LIN {X 0,Y 418.224,Z 205.699,A -85,B 0,C 180,E1 -10122.319,E2 -10122.319} C_VEL
LIN {X 0,Y 418.235,Z 205.697,A -85,B 0,C 180,E1 -10125.108,E2 -10125.108} C_VEL
LIN {X 0,Y 418.224,Z 205.697,A -85,B 0,C 180,E1 -10127.764,E2 -10127.764} C_VEL
LIN {X 0,Y 418.241,Z 205.702,A -85,B 0,C 180,E1 -10131.556,E2 -10131.556} C_VEL
LIN {X 0,Y 418.228,Z 205.712,A -85,B 0,C 180,E1 -10132.974,E2 -10132.974} C_VEL
LIN {X 0,Y 423.651,Z 221.501,A -85,B 0,C 180,E1 -10135.664,E2 -10135.664} C_VEL
LIN {X 0,Y 426.35,Z 230.16,A -85,B 0,C 180,E1 -10137.028,E2 -10137.028} C_VEL
LIN {X 0,Y 433.959,Z 245.967,A -85,B 0,C 180,E1 -10138.023,E2 -10138.023} C_VEL
LIN {X 0,Y 437.099,Z 265.296,A -85,B 0,C 180,E1 -10138.671,E2 -10138.671} C_VEL
LIN {X 0,Y 433.148,Z 437.708,A -85,B 0,C 180,E1 -10141.719,E2 -10141.719} C_VEL
LIN {X 0,Y 432.221,Z 453.77,A -85,B 0,C 180,E1 -10142.161,E2 -10142.161} C_VEL
LIN {X 0,Y 431.126,Z 469.58,A -85,B 0,C 180,E1 -10142.775,E2 -10142.775} C_VEL
LIN {X 0,Y 429.85,Z 484.792,A -85,B 0,C 180,E1 -10143.541,E2 -10143.541} C_VEL
LIN {X 0,Y 428.366,Z 499.512,A -85,B 0,C 180,E1 -10144.469,E2 -10144.469} C_VEL
LIN {X 0,Y 426.802,Z 513.668,A -85,B 0,C 180,E1 -10145.559,E2 -10145.559} C_VEL
LIN {X 0,Y 425.173,Z 527.972,A -85,B 0,C 180,E1 -10146.883,E2 -10146.883} C_VEL
LIN {X 0,Y 423.786,Z 539.159,A -85,B 0,C 180,E1 -10148.092,E2 -10148.092} C_VEL
LIN {X 0,Y 422.302,Z 550.643,A -85,B 0,C 180,E1 -10149.543,E2 -10149.543} C_VEL
LIN {X 0,Y 420.912,Z 562.204,A -85,B 0,C 180,E1 -10151.25,E2 -10151.25} C_VEL
LIN {X 0,Y 419.814,Z 572.306,A -85,B 0,C 180,E1 -10152.997,E2 -10152.997} C_VEL
LIN {X 0,Y 418.809,Z 581.69,A -85,B 0,C 180,E1 -10154.922,E2 -10154.922} C_VEL
LIN {X 0,Y 418.116,Z 589.681,A -85,B 0,C 180,E1 -10156.878,E2 -10156.878} C_VEL
LIN {X 0,Y 417.594,Z 596.384,A -85,B 0,C 180,E1 -10158.839,E2 -10158.839} C_VEL
LIN {X 0,Y 417.237,Z 601.811,A -85,B 0,C 180,E1 -10160.79,E2 -10160.79} C_VEL
LIN {X 0,Y 417.142,Z 605.169,A -85,B 0,C 180,E1 -10162.252,E2 -10162.252} C_VEL
LIN {X 0,Y 417.065,Z 608.619,A -85,B 0,C 180,E1 -10164.195,E2 -10164.195} C_VEL
LIN {X 0,Y 416.965,Z 611.127,A -85,B 0,C 180,E1 -10166.132,E2 -10166.132} C_VEL
LIN {X 0,Y 417.062,Z 612.548,A -85,B 0,C 180,E1 -10168.066,E2 -10168.066} C_VEL
LIN {X 0,Y 416.999,Z 613.082,A -85,B 0,C 180,E1 -10169.998,E2 -10169.998} C_VEL
LIN {X 0,Y 417.061,Z 612.552,A -85,B 0,C 180,E1 -10171.929,E2 -10171.929} C_VEL
LIN {X 0,Y 416.964,Z 611.13,A -85,B 0,C 180,E1 -10173.863,E2 -10173.863} C_VEL
LIN {X 0,Y 417.135,Z 607.929,A -85,B 0,C 180,E1 -10176.259,E2 -10176.259} C_VEL
LIN {X 0,Y 417.18,Z 604.08,A -85,B 0,C 180,E1 -10178.23,E2 -10178.23} C_VEL
LIN {X 0,Y 417.386,Z 599.247,A -85,B 0,C 180,E1 -10180.181,E2 -10180.181} C_VEL
LIN {X 0,Y 417.854,Z 593.155,A -85,B 0,C 180,E1 -10182.134,E2 -10182.134} C_VEL
LIN {X 0,Y 418.386,Z 585.778,A -85,B 0,C 180,E1 -10184.094,E2 -10184.094} C_VEL
LIN {X 0,Y 419.336,Z 576.968,A -85,B 0,C 180,E1 -10186.051,E2 -10186.051} C_VEL
LIN {X 0,Y 420.386,Z 566.446,A -85,B 0,C 180,E1 -10188.013,E2 -10188.013} C_VEL
LIN {X 0,Y 421.704,Z 555.505,A -85,B 0,C 180,E1 -10189.72,E2 -10189.72} C_VEL
LIN {X 0,Y 422.98,Z 544.609,A -85,B 0,C 180,E1 -10191.182,E2 -10191.182} C_VEL
LIN {X 0,Y 424.434,Z 531.99,A -85,B 0,C 180,E1 -10192.639,E2 -10192.639} C_VEL
LIN {X 0,Y 426.083,Z 518.332,A -85,B 0,C 180,E1 -10193.961,E2 -10193.961} C_VEL
LIN {X 0,Y 427.557,Z 505.031,A -85,B 0,C 180,E1 -10195.037,E2 -10195.037} C_VEL
LIN {X 0,Y 429.007,Z 490.343,A -85,B 0,C 180,E1 -10196.032,E2 -10196.032} C_VEL
LIN {X 0,Y 430.365,Z 474.899,A -85,B 0,C 180,E1 -10196.878,E2 -10196.878} C_VEL
LIN {X 0,Y 431.56,Z 458.018,A -85,B 0,C 180,E1 -10197.584,E2 -10197.584} C_VEL
LIN {X 0,Y 432.467,Z 442.335,A -85,B 0,C 180,E1 -10198.048,E2 -10198.048} C_VEL
LIN {X 0,Y 433.152,Z 419.903,A -85,B 0,C 180,E1 -10198.483,E2 -10198.483} C_VEL
LIN {X 0,Y 436.397,Z 265.424,A -85,B 0,C 180,E1 -10201.171,E2 -10201.171} C_VEL
LIN {X 0,Y 432.877,Z 244.923,A -85,B 0,C 180,E1 -10201.839,E2 -10201.839} C_VEL
LIN {X 0,Y 426.312,Z 230.881,A -85,B 0,C 180,E1 -10202.655,E2 -10202.655} C_VEL
LIN {X 0,Y 421.2,Z 214.684,A -85,B 0,C 180,E1 -10205.156,E2 -10205.156} C_VEL
LIN {X 0,Y 418.222,Z 205.707,A -85,B 0,C 180,E1 -10206.617,E2 -10206.617} C_VEL
LIN {X 0,Y 418.225,Z 205.697,A -85,B 0,C 180,E1 -10209.68,E2 -10209.68} C_VEL
LIN {X 0,Y 418.208,Z 205.699,A -85,B 0,C 180,E1 -10212.318,E2 -10212.318} C_VEL
LIN {X 0,Y 418.217,Z 205.698,A -85,B 0,C 180,E1 -10215.107,E2 -10215.107} C_VEL
LIN {X 0,Y 418.235,Z 205.7,A -85,B 0,C 180,E1 -10217.767,E2 -10217.767} C_VEL
LIN {X 0,Y 418.243,Z 205.697,A -85,B 0,C 180,E1 -10220.615,E2 -10220.615} C_VEL
LIN {X 0,Y 418.22,Z 205.694,A -85,B 0,C 180,E1 -10223.974,E2 -10223.974} C_VEL
LIN {X 0,Y 418.23,Z 205.691,A -85,B 0,C 180,E1 -10227.154,E2 -10227.154} C_VEL
LIN {X 0,Y 418.24,Z 205.704,A -85,B 0,C 180,E1 -10230.894,E2 -10230.894} C_VEL
LIN {X 0,Y 418.241,Z 205.683,A -85,B 0,C 180,E1 -10234.094,E2 -10234.094} C_VEL
LIN {X 0,Y 418.245,Z 205.697,A -85,B 0,C 180,E1 -10237.536,E2 -10237.536} C_VEL
LIN {X 0,Y 418.286,Z 205.673,A -85,B 0,C 180,E1 -10240.365,E2 -10240.365} C_VEL
LIN {X 0,Y 418.285,Z 205.693,A -85,B 0,C 180,E1 -10243.404,E2 -10243.404} C_VEL
LIN {X 0,Y 418.323,Z 205.665,A -85,B 0,C 180,E1 -10246.993,E2 -10246.993} C_VEL
LIN {X 0,Y 418.33,Z 205.681,A -85,B 0,C 180,E1 -10250.329,E2 -10250.329} C_VEL
LIN {X 0,Y 418.463,Z 205.666,A -85,B 0,C 180,E1 -10253.249,E2 -10253.249} C_VEL
LIN {X 0,Y 418.312,Z 205.667,A -85,B 0,C 180,E1 -10255.182,E2 -10255.182} C_VEL
LIN {X 0,Y 418.513,Z 205.648,A -85,B 0,C 180,E1 -10258.076,E2 -10258.076} C_VEL
LIN {X 0,Y 418.64,Z 205.645,A -85,B 0,C 180,E1 -10260,E2 -10260} C_VEL
LIN {X 0,Y 418.478,Z 205.661,A -85,B 0,C 180,E1 -10262.888,E2 -10262.888} C_VEL
LIN {X 0,Y 418.461,Z 205.67,A -85,B 0,C 180,E1 -10266.752,E2 -10266.752} C_VEL
LIN {X 0,Y 418.31,Z 205.684,A -85,B 0,C 180,E1 -10269.673,E2 -10269.673} C_VEL
LIN {X 0,Y 418.315,Z 205.682,A -85,B 0,C 180,E1 -10273.002,E2 -10273.002} C_VEL
LIN {X 0,Y 418.291,Z 205.687,A -85,B 0,C 180,E1 -10276.74,E2 -10276.74} C_VEL
LIN {X 0,Y 418.242,Z 205.684,A -85,B 0,C 180,E1 -10279.792,E2 -10279.792} C_VEL
LIN {X 0,Y 418.211,Z 205.702,A -85,B 0,C 180,E1 -10282.738,E2 -10282.738} C_VEL
LIN {X 0,Y 418.244,Z 205.683,A -85,B 0,C 180,E1 -10285.906,E2 -10285.906} C_VEL
LIN {X 0,Y 418.24,Z 205.697,A -85,B 0,C 180,E1 -10289.165,E2 -10289.165} C_VEL
LIN {X 0,Y 418.234,Z 205.686,A -85,B 0,C 180,E1 -10292.847,E2 -10292.847} C_VEL
LIN {X 0,Y 418.223,Z 205.705,A -85,B 0,C 180,E1 -10296.241,E2 -10296.241} C_VEL
LIN {X 0,Y 418.222,Z 205.686,A -85,B 0,C 180,E1 -10299.686,E2 -10299.686} C_VEL
LIN {X 0,Y 418.21,Z 205.706,A -85,B 0,C 180,E1 -10302.324,E2 -10302.324} C_VEL
LIN {X 0,Y 418.218,Z 205.687,A -85,B 0,C 180,E1 -10305.112,E2 -10305.112} C_VEL
LIN {X 0,Y 418.218,Z 205.702,A -85,B 0,C 180,E1 -10307.769,E2 -10307.769} C_VEL
LIN {X 0,Y 418.233,Z 205.693,A -85,B 0,C 180,E1 -10311.561,E2 -10311.561} C_VEL
LIN {X 0,Y 418.248,Z 205.688,A -85,B 0,C 180,E1 -10315.162,E2 -10315.162} C_VEL
LIN {X 0,Y 418.235,Z 205.698,A -85,B 0,C 180,E1 -10317.475,E2 -10317.475} C_VEL
LIN {X 0,Y 418.256,Z 205.694,A -85,B 0,C 180,E1 -10320.9,E2 -10320.9} C_VEL
LIN {X 0,Y 418.228,Z 205.696,A -85,B 0,C 180,E1 -10324.097,E2 -10324.097} C_VEL
LIN {X 0,Y 418.227,Z 205.697,A -85,B 0,C 180,E1 -10327.267,E2 -10327.267} C_VEL
LIN {X 0,Y 418.28,Z 205.691,A -85,B 0,C 180,E1 -10330.367,E2 -10330.367} C_VEL
LIN {X 0,Y 418.277,Z 205.693,A -85,B 0,C 180,E1 -10333.406,E2 -10333.406} C_VEL
LIN {X 0,Y 418.347,Z 205.686,A -85,B 0,C 180,E1 -10337.002,E2 -10337.002} C_VEL
LIN {X 0,Y 418.336,Z 205.686,A -85,B 0,C 180,E1 -10340.331,E2 -10340.331} C_VEL
LIN {X 0,Y 418.455,Z 205.75,A -85,B 0,C 180,E1 -10343.108,E2 -10343.108} C_VEL
LIN {X 0,Y 419.99,Z 210.519,A -85,B 0,C 180,E1 -10343.895,E2 -10343.895} C_VEL
LIN {X 0,Y 432.553,Z 235.499,A -85,B 0,C 180,E1 -10345.43,E2 -10345.43} C_VEL
LIN {X 0,Y 436.628,Z 244.415,A -85,B 0,C 180,E1 -10345.921,E2 -10345.921} C_VEL
LIN {X 0,Y 434.989,Z 317.307,A -85,B 0,C 180,E1 -10347.19,E2 -10347.19} C_VEL
LIN {X 0,Y 434.323,Z 323.153,A -85,B 0,C 180,E1 -10347.252,E2 -10347.252} C_VEL
LIN {X 0,Y 428.84,Z 342.222,A -85,B 0,C 180,E1 -10347.211,E2 -10347.211} C_VEL
LIN {X 0,Y 428.073,Z 348.075,A -85,B 0,C 180,E1 -10347.266,E2 -10347.266} C_VEL
LIN {X 0,Y 426.561,Z 416.445,A -85,B 0,C 180,E1 -10348.498,E2 -10348.498} C_VEL
LIN {X 0,Y 425.738,Z 433.559,A -85,B 0,C 180,E1 -10348.997,E2 -10348.997} C_VEL
LIN {X 0,Y 424.731,Z 449.304,A -85,B 0,C 180,E1 -10349.647,E2 -10349.647} C_VEL
LIN {X 0,Y 423.415,Z 464.949,A -85,B 0,C 180,E1 -10350.478,E2 -10350.478} C_VEL
LIN {X 0,Y 422.031,Z 479.6,A -85,B 0,C 180,E1 -10351.449,E2 -10351.449} C_VEL
LIN {X 0,Y 420.402,Z 494.314,A -85,B 0,C 180,E1 -10352.637,E2 -10352.637} C_VEL
LIN {X 0,Y 418.776,Z 507.961,A -85,B 0,C 180,E1 -10353.972,E2 -10353.972} C_VEL
LIN {X 0,Y 417.194,Z 520.585,A -85,B 0,C 180,E1 -10355.433,E2 -10355.433} C_VEL
LIN {X 0,Y 415.669,Z 532.421,A -85,B 0,C 180,E1 -10357.043,E2 -10357.043} C_VEL
LIN {X 0,Y 414.256,Z 543.314,A -85,B 0,C 180,E1 -10358.785,E2 -10358.785} C_VEL
LIN {X 0,Y 412.951,Z 553.803,A -85,B 0,C 180,E1 -10360.792,E2 -10360.792} C_VEL
LIN {X 0,Y 411.963,Z 562.602,A -85,B 0,C 180,E1 -10362.815,E2 -10362.815} C_VEL
LIN {X 0,Y 411.195,Z 569.983,A -85,B 0,C 180,E1 -10364.857,E2 -10364.857} C_VEL
LIN {X 0,Y 410.629,Z 576.107,A -85,B 0,C 180,E1 -10366.917,E2 -10366.917} C_VEL
LIN {X 0,Y 410.268,Z 580.967,A -85,B 0,C 180,E1 -10368.996,E2 -10368.996} C_VEL
LIN {X 0,Y 409.941,Z 584.701,A -85,B 0,C 180,E1 -10371.103,E2 -10371.103} C_VEL
LIN {X 0,Y 409.767,Z 587.357,A -85,B 0,C 180,E1 -10373.235,E2 -10373.235} C_VEL
LIN {X 0,Y 409.684,Z 588.815,A -85,B 0,C 180,E1 -10375.397,E2 -10375.397} C_VEL
LIN {X 0,Y 409.726,Z 589.143,A -85,B 0,C 180,E1 -10377.591,E2 -10377.591} C_VEL
LIN {X 0,Y 409.785,Z 588.303,A -85,B 0,C 180,E1 -10379.827,E2 -10379.827} C_VEL
LIN {X 0,Y 409.913,Z 586.13,A -85,B 0,C 180,E1 -10382.108,E2 -10382.108} C_VEL
LIN {X 0,Y 410.164,Z 582.538,A -85,B 0,C 180,E1 -10384.434,E2 -10384.434} C_VEL
LIN {X 0,Y 410.493,Z 578.367,A -85,B 0,C 180,E1 -10386.419,E2 -10386.419} C_VEL
LIN {X 0,Y 411.054,Z 572.44,A -85,B 0,C 180,E1 -10388.627,E2 -10388.627} C_VEL
LIN {X 0,Y 411.708,Z 566.367,A -85,B 0,C 180,E1 -10390.443,E2 -10390.443} C_VEL
LIN {X 0,Y 412.67,Z 557.711,A -85,B 0,C 180,E1 -10392.608,E2 -10392.608} C_VEL
LIN {X 0,Y 413.94,Z 547.818,A -85,B 0,C 180,E1 -10394.652,E2 -10394.652} C_VEL
LIN {X 0,Y 415.348,Z 537.429,A -85,B 0,C 180,E1 -10396.459,E2 -10396.459} C_VEL
LIN {X 0,Y 416.979,Z 525.311,A -85,B 0,C 180,E1 -10398.23,E2 -10398.23} C_VEL
LIN {X 0,Y 418.469,Z 513.861,A -85,B 0,C 180,E1 -10399.646,E2 -10399.646} C_VEL
LIN {X 0,Y 420.165,Z 500.476,A -85,B 0,C 180,E1 -10401.059,E2 -10401.059} C_VEL
LIN {X 0,Y 421.909,Z 485.847,A -85,B 0,C 180,E1 -10402.347,E2 -10402.347} C_VEL
LIN {X 0,Y 423.488,Z 471.058,A -85,B 0,C 180,E1 -10403.42,E2 -10403.42} C_VEL
LIN {X 0,Y 424.824,Z 456.217,A -85,B 0,C 180,E1 -10404.286,E2 -10404.286} C_VEL
LIN {X 0,Y 426.038,Z 439.8,A -85,B 0,C 180,E1 -10405.037,E2 -10405.037} C_VEL
LIN {X 0,Y 426.972,Z 423.004,A -85,B 0,C 180,E1 -10405.599,E2 -10405.599} C_VEL
LIN {X 0,Y 427.604,Z 405.792,A -85,B 0,C 180,E1 -10405.978,E2 -10405.978} C_VEL
LIN {X 0,Y 431.375,Z 247.088,A -85,B 0,C 180,E1 -10408.816,E2 -10408.816} C_VEL
LIN {X 0,Y 422.843,Z 229.659,A -85,B 0,C 180,E1 -10409.944,E2 -10409.944} C_VEL
LIN {X 0,Y 414.377,Z 214.394,A -85,B 0,C 180,E1 -10411.094,E2 -10411.094} C_VEL
LIN {X 0,Y 412.834,Z 211.442,A -85,B 0,C 180,E1 -10411.323,E2 -10411.323} C_VEL
LIN {X 0,Y 411.25,Z 206.571,A -85,B 0,C 180,E1 -10412.279,E2 -10412.279} C_VEL
LIN {X 0,Y 411.215,Z 206.574,A -85,B 0,C 180,E1 -10415.783,E2 -10415.783} C_VEL
LIN {X 0,Y 411.199,Z 206.57,A -85,B 0,C 180,E1 -10418.965,E2 -10418.965} C_VEL
LIN {X 0,Y 411.255,Z 206.562,A -85,B 0,C 180,E1 -10422.084,E2 -10422.084} C_VEL
LIN {X 0,Y 411.261,Z 206.567,A -85,B 0,C 180,E1 -10425.147,E2 -10425.147} C_VEL
LIN {X 0,Y 411.284,Z 206.569,A -85,B 0,C 180,E1 -10428.167,E2 -10428.167} C_VEL
LIN {X 0,Y 411.426,Z 206.55,A -85,B 0,C 180,E1 -10432.206,E2 -10432.206} C_VEL
LIN {X 0,Y 411.474,Z 206.541,A -85,B 0,C 180,E1 -10434.117,E2 -10434.117} C_VEL
LIN {X 0,Y 411.51,Z 206.538,A -85,B 0,C 180,E1 -10438.042,E2 -10438.042} C_VEL
LIN {X 0,Y 411.639,Z 206.524,A -85,B 0,C 180,E1 -10439.999,E2 -10439.999} C_VEL
LIN {X 0,Y 411.455,Z 206.543,A -85,B 0,C 180,E1 -10442.937,E2 -10442.937} C_VEL
LIN {X 0,Y 411.464,Z 206.545,A -85,B 0,C 180,E1 -10445.882,E2 -10445.882} C_VEL
LIN {X 0,Y 411.319,Z 206.561,A -85,B 0,C 180,E1 -10448.845,E2 -10448.845} C_VEL
LIN {X 0,Y 411.283,Z 206.567,A -85,B 0,C 180,E1 -10451.832,E2 -10451.832} C_VEL
LIN {X 0,Y 411.259,Z 206.569,A -85,B 0,C 180,E1 -10454.852,E2 -10454.852} C_VEL
LIN {X 0,Y 411.245,Z 206.569,A -85,B 0,C 180,E1 -10457.915,E2 -10457.915} C_VEL
LIN {X 0,Y 411.196,Z 206.578,A -85,B 0,C 180,E1 -10461.034,E2 -10461.034} C_VEL
LIN {X 0,Y 411.218,Z 206.569,A -85,B 0,C 180,E1 -10464.215,E2 -10464.215} C_VEL
LIN {X 0,Y 411.26,Z 206.568,A -85,B 0,C 180,E1 -10467.477,E2 -10467.477} C_VEL
LIN {X 0,Y 411.189,Z 206.579,A -85,B 0,C 180,E1 -10470.847,E2 -10470.847} C_VEL
LIN {X 0,Y 411.193,Z 206.574,A -85,B 0,C 180,E1 -10474.334,E2 -10474.334} C_VEL
LIN {X 0,Y 411.192,Z 206.576,A -85,B 0,C 180,E1 -10477.973,E2 -10477.973} C_VEL
LIN {X 0,Y 411.161,Z 206.573,A -85,B 0,C 180,E1 -10481.227,E2 -10481.227} C_VEL
LIN {X 0,Y 411.175,Z 206.574,A -85,B 0,C 180,E1 -10484.49,E2 -10484.49} C_VEL
LIN {X 0,Y 411.165,Z 206.578,A -85,B 0,C 180,E1 -10488.192,E2 -10488.192} C_VEL
LIN {X 0,Y 411.197,Z 206.577,A -85,B 0,C 180,E1 -10491.832,E2 -10491.832} C_VEL
LIN {X 0,Y 411.219,Z 206.749,A -85,B 0,C 180,E1 -10492.365,E2 -10492.365} C_VEL
LIN {X 0,Y 416.965,Z 223.279,A -85,B 0,C 180,E1 -10495.269,E2 -10495.269} C_VEL
LIN {X 0,Y 419.14,Z 230.129,A -85,B 0,C 180,E1 -10496.353,E2 -10496.353} C_VEL
LIN {X 0,Y 427.046,Z 246.152,A -85,B 0,C 180,E1 -10497.422,E2 -10497.422} C_VEL
LIN {X 0,Y 428.433,Z 249.802,A -85,B 0,C 180,E1 -10497.619,E2 -10497.619} C_VEL
LIN {X 0,Y 431.099,Z 267.046,A -85,B 0,C 180,E1 -10498.201,E2 -10498.201} C_VEL
LIN {X 0,Y 426.953,Z 437.436,A -85,B 0,C 180,E1 -10501.254,E2 -10501.254} C_VEL
LIN {X 0,Y 425.967,Z 453.95,A -85,B 0,C 180,E1 -10501.716,E2 -10501.716} C_VEL
LIN {X 0,Y 424.822,Z 469.64,A -85,B 0,C 180,E1 -10502.337,E2 -10502.337} C_VEL
LIN {X 0,Y 423.497,Z 484.763,A -85,B 0,C 180,E1 -10503.113,E2 -10503.113} C_VEL
LIN {X 0,Y 421.832,Z 500.369,A -85,B 0,C 180,E1 -10504.115,E2 -10504.115} C_VEL
LIN {X 0,Y 420.112,Z 514.978,A -85,B 0,C 180,E1 -10505.276,E2 -10505.276} C_VEL
LIN {X 0,Y 418.429,Z 529.014,A -85,B 0,C 180,E1 -10506.62,E2 -10506.62} C_VEL
LIN {X 0,Y 416.945,Z 540.466,A -85,B 0,C 180,E1 -10507.898,E2 -10507.898} C_VEL
LIN {X 0,Y 415.348,Z 552.287,A -85,B 0,C 180,E1 -10509.443,E2 -10509.443} C_VEL
LIN {X 0,Y 413.918,Z 563.541,A -85,B 0,C 180,E1 -10511.178,E2 -10511.178} C_VEL
LIN {X 0,Y 412.789,Z 573.36,A -85,B 0,C 180,E1 -10512.95,E2 -10512.95} C_VEL
LIN {X 0,Y 411.749,Z 582.616,A -85,B 0,C 180,E1 -10514.91,E2 -10514.91} C_VEL
LIN {X 0,Y 410.989,Z 591.343,A -85,B 0,C 180,E1 -10517.154,E2 -10517.154} C_VEL
LIN {X 0,Y 410.324,Z 599.079,A -85,B 0,C 180,E1 -10519.637,E2 -10519.637} C_VEL
LIN {X 0,Y 410.079,Z 604.974,A -85,B 0,C 180,E1 -10522.118,E2 -10522.118} C_VEL
LIN {X 0,Y 409.979,Z 608.421,A -85,B 0,C 180,E1 -10524.094,E2 -10524.094} C_VEL
LIN {X 0,Y 409.883,Z 610.927,A -85,B 0,C 180,E1 -10526.065,E2 -10526.065} C_VEL
LIN {X 0,Y 409.971,Z 612.346,A -85,B 0,C 180,E1 -10528.033,E2 -10528.033} C_VEL
LIN {X 0,Y 409.921,Z 612.876,A -85,B 0,C 180,E1 -10529.998,E2 -10529.998} C_VEL
LIN {X 0,Y 409.988,Z 612.343,A -85,B 0,C 180,E1 -10531.962,E2 -10531.962} C_VEL
LIN {X 0,Y 409.881,Z 610.915,A -85,B 0,C 180,E1 -10533.93,E2 -10533.93} C_VEL
LIN {X 0,Y 410.037,Z 607.925,A -85,B 0,C 180,E1 -10536.222,E2 -10536.222} C_VEL
LIN {X 0,Y 410.091,Z 603.851,A -85,B 0,C 180,E1 -10538.373,E2 -10538.373} C_VEL
LIN {X 0,Y 410.322,Z 599.008,A -85,B 0,C 180,E1 -10540.358,E2 -10540.358} C_VEL
LIN {X 0,Y 410.836,Z 592.91,A -85,B 0,C 180,E1 -10542.344,E2 -10542.344} C_VEL
LIN {X 0,Y 411.388,Z 585.521,A -85,B 0,C 180,E1 -10544.339,E2 -10544.339} C_VEL
LIN {X 0,Y 412.409,Z 576.698,A -85,B 0,C 180,E1 -10546.328,E2 -10546.328} C_VEL
LIN {X 0,Y 413.495,Z 566.161,A -85,B 0,C 180,E1 -10548.324,E2 -10548.324} C_VEL
LIN {X 0,Y 414.919,Z 555.209,A -85,B 0,C 180,E1 -10550.056,E2 -10550.056} C_VEL
LIN {X 0,Y 416.271,Z 544.283,A -85,B 0,C 180,E1 -10551.54,E2 -10551.54} C_VEL
LIN {X 0,Y 417.832,Z 531.625,A -85,B 0,C 180,E1 -10553.018,E2 -10553.018} C_VEL
LIN {X 0,Y 419.506,Z 517.933,A -85,B 0,C 180,E1 -10554.361,E2 -10554.361} C_VEL
LIN {X 0,Y 421.228,Z 502.917,A -85,B 0,C 180,E1 -10555.578,E2 -10555.578} C_VEL
LIN {X 0,Y 422.756,Z 487.631,A -85,B 0,C 180,E1 -10556.593,E2 -10556.593} C_VEL
LIN {X 0,Y 424.19,Z 471.683,A -85,B 0,C 180,E1 -10557.435,E2 -10557.435} C_VEL
LIN {X 0,Y 425.317,Z 455.528,A -85,B 0,C 180,E1 -10558.091,E2 -10558.091} C_VEL
LIN {X 0,Y 426.294,Z 439.16,A -85,B 0,C 180,E1 -10558.558,E2 -10558.558} C_VEL
LIN {X 0,Y 427.391,Z 389.53,A -85,B 0,C 180,E1 -10559.459,E2 -10559.459} C_VEL
LIN {X 0,Y 430.199,Z 265.695,A -85,B 0,C 180,E1 -10561.644,E2 -10561.644} C_VEL
LIN {X 0,Y 427.058,Z 247.804,A -85,B 0,C 180,E1 -10562.247,E2 -10562.247} C_VEL
LIN {X 0,Y 418.931,Z 230.448,A -85,B 0,C 180,E1 -10563.305,E2 -10563.305} C_VEL
LIN {X 0,Y 413.857,Z 214.643,A -85,B 0,C 180,E1 -10565.82,E2 -10565.82} C_VEL
LIN {X 0,Y 411.188,Z 206.576,A -85,B 0,C 180,E1 -10567.184,E2 -10567.184} C_VEL
LIN {X 0,Y 411.159,Z 206.578,A -85,B 0,C 180,E1 -10570.502,E2 -10570.502} C_VEL
LIN {X 0,Y 411.152,Z 206.578,A -85,B 0,C 180,E1 -10573.131,E2 -10573.131} C_VEL
LIN {X 0,Y 411.15,Z 206.576,A -85,B 0,C 180,E1 -10575.878,E2 -10575.878} C_VEL
LIN {X 0,Y 411.177,Z 206.574,A -85,B 0,C 180,E1 -10578.763,E2 -10578.763} C_VEL
LIN {X 0,Y 411.178,Z 206.577,A -85,B 0,C 180,E1 -10582.025,E2 -10582.025} C_VEL
LIN {X 0,Y 411.179,Z 206.578,A -85,B 0,C 180,E1 -10585.664,E2 -10585.664} C_VEL
LIN {X 0,Y 411.161,Z 206.574,A -85,B 0,C 180,E1 -10589.151,E2 -10589.151} C_VEL
LIN {X 0,Y 411.23,Z 206.567,A -85,B 0,C 180,E1 -10592.521,E2 -10592.521} C_VEL
LIN {X 0,Y 411.2,Z 206.574,A -85,B 0,C 180,E1 -10595.783,E2 -10595.783} C_VEL
LIN {X 0,Y 411.208,Z 206.562,A -85,B 0,C 180,E1 -10598.967,E2 -10598.967} C_VEL
LIN {X 0,Y 411.221,Z 206.565,A -85,B 0,C 180,E1 -10602.084,E2 -10602.084} C_VEL
LIN {X 0,Y 411.231,Z 206.567,A -85,B 0,C 180,E1 -10605.147,E2 -10605.147} C_VEL
LIN {X 0,Y 411.269,Z 206.538,A -85,B 0,C 180,E1 -10608.167,E2 -10608.167} C_VEL
LIN {X 0,Y 411.411,Z 206.549,A -85,B 0,C 180,E1 -10612.186,E2 -10612.186} C_VEL
LIN {X 0,Y 411.459,Z 206.537,A -85,B 0,C 180,E1 -10614.118,E2 -10614.118} C_VEL
LIN {X 0,Y 411.482,Z 206.523,A -85,B 0,C 180,E1 -10618.043,E2 -10618.043} C_VEL
LIN {X 0,Y 411.61,Z 206.521,A -85,B 0,C 180,E1 -10620.001,E2 -10620.001} C_VEL
LIN {X 0,Y 411.434,Z 206.538,A -85,B 0,C 180,E1 -10622.938,E2 -10622.938} C_VEL
LIN {X 0,Y 411.425,Z 206.548,A -85,B 0,C 180,E1 -10626.868,E2 -10626.868} C_VEL
LIN {X 0,Y 411.262,Z 206.562,A -85,B 0,C 180,E1 -10629.84,E2 -10629.84} C_VEL
LIN {X 0,Y 411.275,Z 206.56,A -85,B 0,C 180,E1 -10633.105,E2 -10633.105} C_VEL
LIN {X 0,Y 411.235,Z 206.564,A -85,B 0,C 180,E1 -10636.871,E2 -10636.871} C_VEL
LIN {X 0,Y 411.202,Z 206.561,A -85,B 0,C 180,E1 -10639.989,E2 -10639.989} C_VEL
LIN {X 0,Y 411.176,Z 206.575,A -85,B 0,C 180,E1 -10643.15,E2 -10643.15} C_VEL
LIN {X 0,Y 411.212,Z 206.56,A -85,B 0,C 180,E1 -10646.383,E2 -10646.383} C_VEL
LIN {X 0,Y 411.175,Z 206.578,A -85,B 0,C 180,E1 -10649.715,E2 -10649.715} C_VEL
LIN {X 0,Y 411.183,Z 206.564,A -85,B 0,C 180,E1 -10653.159,E2 -10653.159} C_VEL
LIN {X 0,Y 411.171,Z 206.58,A -85,B 0,C 180,E1 -10656.555,E2 -10656.555} C_VEL
LIN {X 0,Y 411.187,Z 206.562,A -85,B 0,C 180,E1 -10659.73,E2 -10659.73} C_VEL
LIN {X 0,Y 411.155,Z 206.579,A -85,B 0,C 180,E1 -10663.137,E2 -10663.137} C_VEL
LIN {X 0,Y 411.15,Z 206.57,A -85,B 0,C 180,E1 -10665.884,E2 -10665.884} C_VEL
LIN {X 0,Y 411.142,Z 206.58,A -85,B 0,C 180,E1 -10668.776,E2 -10668.776} C_VEL
LIN {X 0,Y 411.18,Z 206.576,A -85,B 0,C 180,E1 -10672.029,E2 -10672.029} C_VEL
LIN {X 0,Y 411.195,Z 206.567,A -85,B 0,C 180,E1 -10675.67,E2 -10675.67} C_VEL
LIN {X 0,Y 411.18,Z 206.575,A -85,B 0,C 180,E1 -10679.156,E2 -10679.156} C_VEL
LIN {X 0,Y 411.181,Z 206.578,A -85,B 0,C 180,E1 -10682.521,E2 -10682.521} C_VEL
LIN {X 0,Y 411.198,Z 206.578,A -85,B 0,C 180,E1 -10685.786,E2 -10685.786} C_VEL
LIN {X 0,Y 411.192,Z 206.577,A -85,B 0,C 180,E1 -10688.969,E2 -10688.969} C_VEL
LIN {X 0,Y 411.227,Z 206.578,A -85,B 0,C 180,E1 -10692.087,E2 -10692.087} C_VEL
LIN {X 0,Y 411.231,Z 206.574,A -85,B 0,C 180,E1 -10695.149,E2 -10695.149} C_VEL
LIN {X 0,Y 411.283,Z 206.564,A -85,B 0,C 180,E1 -10698.17,E2 -10698.17} C_VEL
LIN {X 0,Y 411.318,Z 206.564,A -85,B 0,C 180,E1 -10701.157,E2 -10701.157} C_VEL
LIN {X 0,Y 411.414,Z 206.705,A -85,B 0,C 180,E1 -10702.584,E2 -10702.584} C_VEL
LIN {X 0,Y 412.733,Z 210.707,A -85,B 0,C 180,E1 -10703.263,E2 -10703.263} C_VEL
LIN {X 0,Y 426.594,Z 237.914,A -85,B 0,C 180,E1 -10704.998,E2 -10704.998} C_VEL
LIN {X 0,Y 430.444,Z 246.548,A -85,B 0,C 180,E1 -10705.479,E2 -10705.479} C_VEL
LIN {X 0,Y 428.073,Z 348.075,A -85,B 0,C 180,E1 -10707.266,E2 -10707.266} C_VEL
LIN {X 0,Y 427.334,Z 353.923,A -85,B 0,C 180,E1 -10707.324,E2 -10707.324} C_VEL
LIN {X 0,Y 421.952,Z 373.01,A -85,B 0,C 180,E1 -10707.294,E2 -10707.294} C_VEL
LIN {X 0,Y 421.182,Z 378.86,A -85,B 0,C 180,E1 -10707.351,E2 -10707.351} C_VEL
LIN {X 0,Y 420.232,Z 417.941,A -85,B 0,C 180,E1 -10708.086,E2 -10708.086} C_VEL
LIN {X 0,Y 419.394,Z 434.723,A -85,B 0,C 180,E1 -10708.592,E2 -10708.592} C_VEL
LIN {X 0,Y 418.374,Z 449.581,A -85,B 0,C 180,E1 -10709.22,E2 -10709.22} C_VEL
LIN {X 0,Y 417.101,Z 464.231,A -85,B 0,C 180,E1 -10710.002,E2 -10710.002} C_VEL
LIN {X 0,Y 415.54,Z 479.977,A -85,B 0,C 180,E1 -10711.056,E2 -10711.056} C_VEL
LIN {X 0,Y 413.792,Z 495.249,A -85,B 0,C 180,E1 -10712.314,E2 -10712.314} C_VEL
LIN {X 0,Y 412.078,Z 508.809,A -85,B 0,C 180,E1 -10713.669,E2 -10713.669} C_VEL
LIN {X 0,Y 410.493,Z 520.988,A -85,B 0,C 180,E1 -10715.111,E2 -10715.111} C_VEL
LIN {X 0,Y 408.968,Z 532.258,A -85,B 0,C 180,E1 -10716.663,E2 -10716.663} C_VEL
LIN {X 0,Y 407.477,Z 543.191,A -85,B 0,C 180,E1 -10718.432,E2 -10718.432} C_VEL
LIN {X 0,Y 406.239,Z 552.492,A -85,B 0,C 180,E1 -10720.216,E2 -10720.216} C_VEL
LIN {X 0,Y 405.125,Z 561.571,A -85,B 0,C 180,E1 -10722.271,E2 -10722.271} C_VEL
LIN {X 0,Y 404.414,Z 568.327,A -85,B 0,C 180,E1 -10724.083,E2 -10724.083} C_VEL
LIN {X 0,Y 403.714,Z 574.732,A -85,B 0,C 180,E1 -10726.175,E2 -10726.175} C_VEL
LIN {X 0,Y 403.296,Z 579.937,A -85,B 0,C 180,E1 -10728.283,E2 -10728.283} C_VEL
LIN {X 0,Y 402.959,Z 584.029,A -85,B 0,C 180,E1 -10730.417,E2 -10730.417} C_VEL
LIN {X 0,Y 402.724,Z 586.912,A -85,B 0,C 180,E1 -10732.579,E2 -10732.579} C_VEL
LIN {X 0,Y 402.619,Z 588.744,A -85,B 0,C 180,E1 -10734.809,E2 -10734.809} C_VEL
LIN {X 0,Y 402.639,Z 589.42,A -85,B 0,C 180,E1 -10737.101,E2 -10737.101} C_VEL
LIN {X 0,Y 402.676,Z 588.842,A -85,B 0,C 180,E1 -10739.256,E2 -10739.256} C_VEL
LIN {X 0,Y 402.783,Z 587.042,A -85,B 0,C 180,E1 -10741.566,E2 -10741.566} C_VEL
LIN {X 0,Y 403.009,Z 583.892,A -85,B 0,C 180,E1 -10743.922,E2 -10743.922} C_VEL
LIN {X 0,Y 403.316,Z 580.508,A -85,B 0,C 180,E1 -10745.716,E2 -10745.716} C_VEL
LIN {X 0,Y 403.827,Z 574.995,A -85,B 0,C 180,E1 -10748.004,E2 -10748.004} C_VEL
LIN {X 0,Y 404.524,Z 568.517,A -85,B 0,C 180,E1 -10750.142,E2 -10750.142} C_VEL
LIN {X 0,Y 405.32,Z 561.241,A -85,B 0,C 180,E1 -10752.103,E2 -10752.103} C_VEL
LIN {X 0,Y 406.493,Z 552.384,A -85,B 0,C 180,E1 -10754.1,E2 -10754.1} C_VEL
LIN {X 0,Y 407.931,Z 542.397,A -85,B 0,C 180,E1 -10755.997,E2 -10755.997} C_VEL
LIN {X 0,Y 409.521,Z 531.204,A -85,B 0,C 180,E1 -10757.798,E2 -10757.798} C_VEL
LIN {X 0,Y 411.295,Z 518.554,A -85,B 0,C 180,E1 -10759.509,E2 -10759.509} C_VEL
LIN {X 0,Y 413.077,Z 505.519,A -85,B 0,C 180,E1 -10760.985,E2 -10760.985} C_VEL
LIN {X 0,Y 414.866,Z 491.509,A -85,B 0,C 180,E1 -10762.319,E2 -10762.319} C_VEL
LIN {X 0,Y 416.56,Z 476.984,A -85,B 0,C 180,E1 -10763.467,E2 -10763.467} C_VEL
LIN {X 0,Y 418.05,Z 462.403,A -85,B 0,C 180,E1 -10764.416,E2 -10764.416} C_VEL
LIN {X 0,Y 419.333,Z 446.948,A -85,B 0,C 180,E1 -10765.21,E2 -10765.21} C_VEL
LIN {X 0,Y 420.417,Z 430.767,A -85,B 0,C 180,E1 -10765.84,E2 -10765.84} C_VEL
LIN {X 0,Y 421.195,Z 413.932,A -85,B 0,C 180,E1 -10766.3,E2 -10766.3} C_VEL
LIN {X 0,Y 425.399,Z 249.363,A -85,B 0,C 180,E1 -10769.298,E2 -10769.298} C_VEL
LIN {X 0,Y 416.772,Z 231.707,A -85,B 0,C 180,E1 -10770.48,E2 -10770.48} C_VEL
LIN {X 0,Y 409.26,Z 218.266,A -85,B 0,C 180,E1 -10771.53,E2 -10771.53} C_VEL
LIN {X 0,Y 405.527,Z 211.622,A -85,B 0,C 180,E1 -10772.1,E2 -10772.1} C_VEL
LIN {X 0,Y 404.219,Z 207.447,A -85,B 0,C 180,E1 -10772.949,E2 -10772.949} C_VEL
LIN {X 0,Y 404.174,Z 207.456,A -85,B 0,C 180,E1 -10775.334,E2 -10775.334} C_VEL
LIN {X 0,Y 404.141,Z 207.452,A -85,B 0,C 180,E1 -10778.58,E2 -10778.58} C_VEL
LIN {X 0,Y 404.213,Z 207.442,A -85,B 0,C 180,E1 -10781.761,E2 -10781.761} C_VEL
LIN {X 0,Y 404.208,Z 207.446,A -85,B 0,C 180,E1 -10784.882,E2 -10784.882} C_VEL
LIN {X 0,Y 404.257,Z 207.443,A -85,B 0,C 180,E1 -10787.958,E2 -10787.958} C_VEL
LIN {X 0,Y 404.404,Z 207.424,A -85,B 0,C 180,E1 -10792.132,E2 -10792.132} C_VEL
LIN {X 0,Y 404.422,Z 207.419,A -85,B 0,C 180,E1 -10794.015,E2 -10794.015} C_VEL
LIN {X 0,Y 404.479,Z 207.414,A -85,B 0,C 180,E1 -10798.008,E2 -10798.008} C_VEL
LIN {X 0,Y 404.609,Z 207.4,A -85,B 0,C 180,E1 -10799.999,E2 -10799.999} C_VEL
LIN {X 0,Y 404.414,Z 207.421,A -85,B 0,C 180,E1 -10802.988,E2 -10802.988} C_VEL
LIN {X 0,Y 404.412,Z 207.423,A -85,B 0,C 180,E1 -10805.985,E2 -10805.985} C_VEL
LIN {X 0,Y 404.266,Z 207.44,A -85,B 0,C 180,E1 -10809.001,E2 -10809.001} C_VEL
LIN {X 0,Y 404.256,Z 207.44,A -85,B 0,C 180,E1 -10812.041,E2 -10812.041} C_VEL
LIN {X 0,Y 404.205,Z 207.45,A -85,B 0,C 180,E1 -10815.118,E2 -10815.118} C_VEL
LIN {X 0,Y 404.204,Z 207.445,A -85,B 0,C 180,E1 -10818.238,E2 -10818.238} C_VEL
LIN {X 0,Y 404.138,Z 207.454,A -85,B 0,C 180,E1 -10821.419,E2 -10821.419} C_VEL
LIN {X 0,Y 404.174,Z 207.447,A -85,B 0,C 180,E1 -10824.665,E2 -10824.665} C_VEL
LIN {X 0,Y 404.196,Z 207.448,A -85,B 0,C 180,E1 -10827.999,E2 -10827.999} C_VEL
LIN {X 0,Y 404.139,Z 207.454,A -85,B 0,C 180,E1 -10831.557,E2 -10831.557} C_VEL
LIN {X 0,Y 404.179,Z 207.451,A -85,B 0,C 180,E1 -10835.016,E2 -10835.016} C_VEL
LIN {X 0,Y 404.151,Z 207.454,A -85,B 0,C 180,E1 -10838.757,E2 -10838.757} C_VEL
LIN {X 0,Y 404.119,Z 207.45,A -85,B 0,C 180,E1 -10841.598,E2 -10841.598} C_VEL
LIN {X 0,Y 404.145,Z 207.45,A -85,B 0,C 180,E1 -10844.521,E2 -10844.521} C_VEL
LIN {X 0,Y 404.125,Z 207.454,A -85,B 0,C 180,E1 -10847.293,E2 -10847.293} C_VEL
LIN {X 0,Y 404.134,Z 207.454,A -85,B 0,C 180,E1 -10849.95,E2 -10849.95} C_VEL
LIN {X 0,Y 404.147,Z 207.493,A -85,B 0,C 180,E1 -10851.673,E2 -10851.673} C_VEL
LIN {X 0,Y 409.706,Z 223.387,A -85,B 0,C 180,E1 -10854.566,E2 -10854.566} C_VEL
LIN {X 0,Y 411.788,Z 229.649,A -85,B 0,C 180,E1 -10855.619,E2 -10855.619} C_VEL
LIN {X 0,Y 420.77,Z 247.691,A -85,B 0,C 180,E1 -10856.879,E2 -10856.879} C_VEL
LIN {X 0,Y 422.715,Z 252.19,A -85,B 0,C 180,E1 -10857.154,E2 -10857.154} C_VEL
LIN {X 0,Y 425.138,Z 267.569,A -85,B 0,C 180,E1 -10857.691,E2 -10857.691} C_VEL
LIN {X 0,Y 420.747,Z 438.039,A -85,B 0,C 180,E1 -10860.795,E2 -10860.795} C_VEL
LIN {X 0,Y 419.676,Z 455.034,A -85,B 0,C 180,E1 -10861.287,E2 -10861.287} C_VEL
LIN {X 0,Y 418.44,Z 470.996,A -85,B 0,C 180,E1 -10861.946,E2 -10861.946} C_VEL
LIN {X 0,Y 416.935,Z 486.741,A -85,B 0,C 180,E1 -10862.79,E2 -10862.79} C_VEL
LIN {X 0,Y 415.336,Z 501.097,A -85,B 0,C 180,E1 -10863.743,E2 -10863.743} C_VEL
LIN {X 0,Y 413.462,Z 516.343,A -85,B 0,C 180,E1 -10864.985,E2 -10864.985} C_VEL
LIN {X 0,Y 411.687,Z 530.084,A -85,B 0,C 180,E1 -10866.347,E2 -10866.347} C_VEL
LIN {X 0,Y 410.024,Z 542.178,A -85,B 0,C 180,E1 -10867.756,E2 -10867.756} C_VEL
LIN {X 0,Y 408.379,Z 553.87,A -85,B 0,C 180,E1 -10869.34,E2 -10869.34} C_VEL
LIN {X 0,Y 406.9,Z 564.881,A -85,B 0,C 180,E1 -10871.102,E2 -10871.102} C_VEL
LIN {X 0,Y 405.777,Z 574.289,A -85,B 0,C 180,E1 -10872.874,E2 -10872.874} C_VEL
LIN {X 0,Y 404.67,Z 583.464,A -85,B 0,C 180,E1 -10874.898,E2 -10874.898} C_VEL
LIN {X 0,Y 403.948,Z 591.354,A -85,B 0,C 180,E1 -10876.981,E2 -10876.981} C_VEL
LIN {X 0,Y 403.269,Z 598.888,A -85,B 0,C 180,E1 -10879.454,E2 -10879.454} C_VEL
LIN {X 0,Y 402.998,Z 604.779,A -85,B 0,C 180,E1 -10881.978,E2 -10881.978} C_VEL
LIN {X 0,Y 402.896,Z 608.224,A -85,B 0,C 180,E1 -10883.99,E2 -10883.99} C_VEL
LIN {X 0,Y 402.802,Z 610.727,A -85,B 0,C 180,E1 -10885.996,E2 -10885.996} C_VEL
LIN {X 0,Y 402.882,Z 612.145,A -85,B 0,C 180,E1 -10887.998,E2 -10887.998} C_VEL
LIN {X 0,Y 402.846,Z 612.671,A -85,B 0,C 180,E1 -10889.998,E2 -10889.998} C_VEL
LIN {X 0,Y 402.897,Z 612.134,A -85,B 0,C 180,E1 -10891.997,E2 -10891.997} C_VEL
LIN {X 0,Y 402.801,Z 610.7,A -85,B 0,C 180,E1 -10893.999,E2 -10893.999} C_VEL
LIN {X 0,Y 402.934,Z 607.929,A -85,B 0,C 180,E1 -10896.179,E2 -10896.179} C_VEL
LIN {X 0,Y 403.024,Z 603.622,A -85,B 0,C 180,E1 -10898.521,E2 -10898.521} C_VEL
LIN {X 0,Y 403.266,Z 598.769,A -85,B 0,C 180,E1 -10900.541,E2 -10900.541} C_VEL
LIN {X 0,Y 403.794,Z 592.779,A -85,B 0,C 180,E1 -10902.527,E2 -10902.527} C_VEL
LIN {X 0,Y 404.418,Z 585.264,A -85,B 0,C 180,E1 -10904.592,E2 -10904.592} C_VEL
LIN {X 0,Y 405.485,Z 576.42,A -85,B 0,C 180,E1 -10906.614,E2 -10906.614} C_VEL
LIN {X 0,Y 406.488,Z 567.257,A -85,B 0,C 180,E1 -10908.39,E2 -10908.39} C_VEL
LIN {X 0,Y 407.91,Z 556.528,A -85,B 0,C 180,E1 -10910.153,E2 -10910.153} C_VEL
LIN {X 0,Y 409.446,Z 544.749,A -85,B 0,C 180,E1 -10911.807,E2 -10911.807} C_VEL
LIN {X 0,Y 411.052,Z 532.418,A -85,B 0,C 180,E1 -10913.286,E2 -10913.286} C_VEL
LIN {X 0,Y 412.955,Z 517.527,A -85,B 0,C 180,E1 -10914.773,E2 -10914.773} C_VEL
LIN {X 0,Y 414.743,Z 502.465,A -85,B 0,C 180,E1 -10916.008,E2 -10916.008} C_VEL
LIN {X 0,Y 416.281,Z 488.017,A -85,B 0,C 180,E1 -10916.979,E2 -10916.979} C_VEL
LIN {X 0,Y 417.748,Z 472.378,A -85,B 0,C 180,E1 -10917.826,E2 -10917.826} C_VEL
LIN {X 0,Y 418.908,Z 456.587,A -85,B 0,C 180,E1 -10918.492,E2 -10918.492} C_VEL
LIN {X 0,Y 419.988,Z 439.405,A -85,B 0,C 180,E1 -10918.993,E2 -10918.993} C_VEL
LIN {X 0,Y 420.864,Z 402.718,A -85,B 0,C 180,E1 -10919.68,E2 -10919.68} C_VEL
LIN {X 0,Y 424.108,Z 267.724,A -85,B 0,C 180,E1 -10922.09,E2 -10922.09} C_VEL
LIN {X 0,Y 421.28,Z 250.66,A -85,B 0,C 180,E1 -10922.664,E2 -10922.664} C_VEL
LIN {X 0,Y 411.639,Z 230.283,A -85,B 0,C 180,E1 -10923.939,E2 -10923.939} C_VEL
LIN {X 0,Y 406.871,Z 215.688,A -85,B 0,C 180,E1 -10926.326,E2 -10926.326} C_VEL
LIN {X 0,Y 404.134,Z 207.454,A -85,B 0,C 180,E1 -10927.763,E2 -10927.763} C_VEL
LIN {X 0,Y 404.128,Z 207.452,A -85,B 0,C 180,E1 -10930.077,E2 -10930.077} C_VEL
LIN {X 0,Y 404.132,Z 207.452,A -85,B 0,C 180,E1 -10933.081,E2 -10933.081} C_VEL
LIN {X 0,Y 404.13,Z 207.45,A -85,B 0,C 180,E1 -10935.924,E2 -10935.924} C_VEL
LIN {X 0,Y 404.129,Z 207.452,A -85,B 0,C 180,E1 -10938.637,E2 -10938.637} C_VEL
LIN {X 0,Y 404.136,Z 207.457,A -85,B 0,C 180,E1 -10941.489,E2 -10941.489} C_VEL
LIN {X 0,Y 404.159,Z 207.452,A -85,B 0,C 180,E1 -10944.982,E2 -10944.982} C_VEL
LIN {X 0,Y 404.114,Z 207.444,A -85,B 0,C 180,E1 -10948.552,E2 -10948.552} C_VEL
LIN {X 0,Y 404.166,Z 207.449,A -85,B 0,C 180,E1 -10951.999,E2 -10951.999} C_VEL
LIN {X 0,Y 404.149,Z 207.451,A -85,B 0,C 180,E1 -10955.333,E2 -10955.333} C_VEL
LIN {X 0,Y 404.164,Z 207.446,A -85,B 0,C 180,E1 -10958.583,E2 -10958.583} C_VEL
LIN {X 0,Y 404.182,Z 207.441,A -85,B 0,C 180,E1 -10961.761,E2 -10961.761} C_VEL
LIN {X 0,Y 404.176,Z 207.449,A -85,B 0,C 180,E1 -10964.881,E2 -10964.881} C_VEL
LIN {X 0,Y 404.239,Z 207.412,A -85,B 0,C 180,E1 -10967.958,E2 -10967.958} C_VEL
LIN {X 0,Y 404.352,Z 207.428,A -85,B 0,C 180,E1 -10972.008,E2 -10972.008} C_VEL
LIN {X 0,Y 404.405,Z 207.415,A -85,B 0,C 180,E1 -10974.015,E2 -10974.015} C_VEL
LIN {X 0,Y 404.451,Z 207.399,A -85,B 0,C 180,E1 -10978.009,E2 -10978.009} C_VEL
LIN {X 0,Y 404.58,Z 207.397,A -85,B 0,C 180,E1 -10980.001,E2 -10980.001} C_VEL
LIN {X 0,Y 404.391,Z 207.414,A -85,B 0,C 180,E1 -10982.989,E2 -10982.989} C_VEL
LIN {X 0,Y 404.365,Z 207.422,A -85,B 0,C 180,E1 -10986.697,E2 -10986.697} C_VEL
LIN {X 0,Y 404.26,Z 207.437,A -85,B 0,C 180,E1 -10989.002,E2 -10989.002} C_VEL
LIN {X 0,Y 404.226,Z 207.424,A -85,B 0,C 180,E1 -10992.043,E2 -10992.043} C_VEL
LIN {X 0,Y 404.181,Z 207.448,A -85,B 0,C 180,E1 -10995.119,E2 -10995.119} C_VEL
LIN {X 0,Y 404.181,Z 207.436,A -85,B 0,C 180,E1 -10998.24,E2 -10998.24} C_VEL
LIN {X 0,Y 404.111,Z 207.455,A -85,B 0,C 180,E1 -11001.421,E2 -11001.421} C_VEL
LIN {X 0,Y 404.151,Z 207.442,A -85,B 0,C 180,E1 -11004.668,E2 -11004.668} C_VEL
LIN {X 0,Y 404.17,Z 207.446,A -85,B 0,C 180,E1 -11008.002,E2 -11008.002} C_VEL
LIN {X 0,Y 404.115,Z 207.451,A -85,B 0,C 180,E1 -11011.56,E2 -11011.56} C_VEL
LIN {X 0,Y 404.162,Z 207.45,A -85,B 0,C 180,E1 -11015.019,E2 -11015.019} C_VEL
LIN {X 0,Y 404.128,Z 207.441,A -85,B 0,C 180,E1 -11018.761,E2 -11018.761} C_VEL
LIN {X 0,Y 404.103,Z 207.458,A -85,B 0,C 180,E1 -11021.603,E2 -11021.603} C_VEL
LIN {X 0,Y 404.128,Z 207.445,A -85,B 0,C 180,E1 -11024.525,E2 -11024.525} C_VEL
LIN {X 0,Y 404.116,Z 207.456,A -85,B 0,C 180,E1 -11027.298,E2 -11027.298} C_VEL
LIN {X 0,Y 404.12,Z 207.451,A -85,B 0,C 180,E1 -11029.955,E2 -11029.955} C_VEL
LIN {X 0,Y 404.126,Z 207.456,A -85,B 0,C 180,E1 -11033.128,E2 -11033.128} C_VEL
LIN {X 0,Y 404.134,Z 207.449,A -85,B 0,C 180,E1 -11036.191,E2 -11036.191} C_VEL
LIN {X 0,Y 404.136,Z 207.45,A -85,B 0,C 180,E1 -11039.718,E2 -11039.718} C_VEL
LIN {X 0,Y 404.127,Z 207.455,A -85,B 0,C 180,E1 -11043.122,E2 -11043.122} C_VEL
LIN {X 0,Y 404.152,Z 207.453,A -85,B 0,C 180,E1 -11046.428,E2 -11046.428} C_VEL
LIN {X 0,Y 404.188,Z 207.45,A -85,B 0,C 180,E1 -11049.878,E2 -11049.878} C_VEL
LIN {X 0,Y 404.172,Z 207.451,A -85,B 0,C 180,E1 -11053.016,E2 -11053.016} C_VEL
LIN {X 0,Y 404.283,Z 207.438,A -85,B 0,C 180,E1 -11056.942,E2 -11056.942} C_VEL
LIN {X 0,Y 404.255,Z 207.44,A -85,B 0,C 180,E1 -11059.991,E2 -11059.991} C_VEL
LIN {X 0,Y 404.339,Z 207.472,A -85,B 0,C 180,E1 -11062.01,E2 -11062.01} C_VEL
LIN {X 0,Y 405.4,Z 210.83,A -85,B 0,C 180,E1 -11062.595,E2 -11062.595} C_VEL
LIN {X 0,Y 413.163,Z 225.695,A -85,B 0,C 180,E1 -11063.614,E2 -11063.614} C_VEL
LIN {X 0,Y 422.187,Z 243.919,A -85,B 0,C 180,E1 -11064.757,E2 -11064.757} C_VEL
LIN {X 0,Y 424.352,Z 248.675,A -85,B 0,C 180,E1 -11065.029,E2 -11065.029} C_VEL
LIN {X 0,Y 421.182,Z 378.86,A -85,B 0,C 180,E1 -11067.351,E2 -11067.351} C_VEL
LIN {X 0,Y 420.404,Z 384.713,A -85,B 0,C 180,E1 -11067.405,E2 -11067.405} C_VEL
LIN {X 0,Y 414.992,Z 403.791,A -85,B 0,C 180,E1 -11067.37,E2 -11067.37} C_VEL
LIN {X 0,Y 414.274,Z 409.623,A -85,B 0,C 180,E1 -11067.446,E2 -11067.446} C_VEL
LIN {X 0,Y 413.62,Z 425.91,A -85,B 0,C 180,E1 -11067.842,E2 -11067.842} C_VEL
LIN {X 0,Y 412.557,Z 442.559,A -85,B 0,C 180,E1 -11068.447,E2 -11068.447} C_VEL
LIN {X 0,Y 411.305,Z 458.111,A -85,B 0,C 180,E1 -11069.207,E2 -11069.207} C_VEL
LIN {X 0,Y 409.914,Z 472.975,A -85,B 0,C 180,E1 -11070.125,E2 -11070.125} C_VEL
LIN {X 0,Y 408.374,Z 486.599,A -85,B 0,C 180,E1 -11071.144,E2 -11071.144} C_VEL
LIN {X 0,Y 406.521,Z 501.295,A -85,B 0,C 180,E1 -11072.479,E2 -11072.479} C_VEL
LIN {X 0,Y 404.82,Z 513.985,A -85,B 0,C 180,E1 -11073.86,E2 -11073.86} C_VEL
LIN {X 0,Y 403.19,Z 525.804,A -85,B 0,C 180,E1 -11075.365,E2 -11075.365} C_VEL
LIN {X 0,Y 401.564,Z 537.015,A -85,B 0,C 180,E1 -11077.039,E2 -11077.039} C_VEL
LIN {X 0,Y 400.118,Z 547.228,A -85,B 0,C 180,E1 -11078.843,E2 -11078.843} C_VEL
LIN {X 0,Y 398.746,Z 557.188,A -85,B 0,C 180,E1 -11080.924,E2 -11080.924} C_VEL
LIN {X 0,Y 397.859,Z 564.621,A -85,B 0,C 180,E1 -11082.758,E2 -11082.758} C_VEL
LIN {X 0,Y 397.06,Z 571.703,A -85,B 0,C 180,E1 -11084.873,E2 -11084.873} C_VEL
LIN {X 0,Y 396.493,Z 577.098,A -85,B 0,C 180,E1 -11086.827,E2 -11086.827} C_VEL
LIN {X 0,Y 396.089,Z 582.225,A -85,B 0,C 180,E1 -11089.165,E2 -11089.165} C_VEL
LIN {X 0,Y 395.813,Z 584.945,A -85,B 0,C 180,E1 -11090.802,E2 -11090.802} C_VEL
LIN {X 0,Y 395.591,Z 587.662,A -85,B 0,C 180,E1 -11093.009,E2 -11093.009} C_VEL
LIN {X 0,Y 395.51,Z 589.169,A -85,B 0,C 180,E1 -11095.245,E2 -11095.245} C_VEL
LIN {X 0,Y 395.541,Z 589.571,A -85,B 0,C 180,E1 -11097.516,E2 -11097.516} C_VEL
LIN {X 0,Y 395.578,Z 588.801,A -85,B 0,C 180,E1 -11099.834,E2 -11099.834} C_VEL
LIN {X 0,Y 395.75,Z 586.673,A -85,B 0,C 180,E1 -11102.194,E2 -11102.194} C_VEL
LIN {X 0,Y 396.008,Z 583.157,A -85,B 0,C 180,E1 -11104.606,E2 -11104.606} C_VEL
LIN {X 0,Y 396.367,Z 579.574,A -85,B 0,C 180,E1 -11106.442,E2 -11106.442} C_VEL
LIN {X 0,Y 396.996,Z 573.499,A -85,B 0,C 180,E1 -11108.836,E2 -11108.836} C_VEL
LIN {X 0,Y 397.731,Z 567.192,A -85,B 0,C 180,E1 -11110.83,E2 -11110.83} C_VEL
LIN {X 0,Y 398.806,Z 558.626,A -85,B 0,C 180,E1 -11113.07,E2 -11113.07} C_VEL
LIN {X 0,Y 400.155,Z 549.562,A -85,B 0,C 180,E1 -11115.042,E2 -11115.042} C_VEL
LIN {X 0,Y 401.713,Z 538.965,A -85,B 0,C 180,E1 -11116.975,E2 -11116.975} C_VEL
LIN {X 0,Y 403.415,Z 527.724,A -85,B 0,C 180,E1 -11118.703,E2 -11118.703} C_VEL
LIN {X 0,Y 405.275,Z 514.999,A -85,B 0,C 180,E1 -11120.363,E2 -11120.363} C_VEL
LIN {X 0,Y 407.097,Z 502.111,A -85,B 0,C 180,E1 -11121.783,E2 -11121.783} C_VEL
LIN {X 0,Y 408.834,Z 488.864,A -85,B 0,C 180,E1 -11123.01,E2 -11123.01} C_VEL
LIN {X 0,Y 410.472,Z 474.69,A -85,B 0,C 180,E1 -11124.102,E2 -11124.102} C_VEL
LIN {X 0,Y 412.07,Z 459.58,A -85,B 0,C 180,E1 -11125.052,E2 -11125.052} C_VEL
LIN {X 0,Y 413.434,Z 443.669,A -85,B 0,C 180,E1 -11125.844,E2 -11125.844} C_VEL
LIN {X 0,Y 414.504,Z 427.443,A -85,B 0,C 180,E1 -11126.447,E2 -11126.447} C_VEL
LIN {X 0,Y 415.233,Z 411.084,A -85,B 0,C 180,E1 -11126.855,E2 -11126.855} C_VEL
LIN {X 0,Y 419.441,Z 251.509,A -85,B 0,C 180,E1 -11129.802,E2 -11129.802} C_VEL
LIN {X 0,Y 410.761,Z 233.933,A -85,B 0,C 180,E1 -11131.029,E2 -11131.029} C_VEL
LIN {X 0,Y 400.877,Z 216.296,A -85,B 0,C 180,E1 -11132.473,E2 -11132.473} C_VEL
LIN {X 0,Y 398.373,Z 211.951,A -85,B 0,C 180,E1 -11132.875,E2 -11132.875} C_VEL
LIN {X 0,Y 397.124,Z 208.326,A -85,B 0,C 180,E1 -11133.67,E2 -11133.67} C_VEL
LIN {X 0,Y 397.115,Z 208.331,A -85,B 0,C 180,E1 -11136.968,E2 -11136.968} C_VEL
LIN {X 0,Y 397.151,Z 208.328,A -85,B 0,C 180,E1 -11140.352,E2 -11140.352} C_VEL
LIN {X 0,Y 397.169,Z 208.32,A -85,B 0,C 180,E1 -11143.553,E2 -11143.553} C_VEL
LIN {X 0,Y 397.232,Z 208.315,A -85,B 0,C 180,E1 -11146.702,E2 -11146.702} C_VEL
LIN {X 0,Y 397.218,Z 208.318,A -85,B 0,C 180,E1 -11149.808,E2 -11149.808} C_VEL
LIN {X 0,Y 397.351,Z 208.301,A -85,B 0,C 180,E1 -11152.887,E2 -11152.887} C_VEL
LIN {X 0,Y 397.253,Z 208.313,A -85,B 0,C 180,E1 -11154.925,E2 -11154.925} C_VEL
LIN {X 0,Y 397.448,Z 208.29,A -85,B 0,C 180,E1 -11157.973,E2 -11157.973} C_VEL
LIN {X 0,Y 397.578,Z 208.276,A -85,B 0,C 180,E1 -11159.999,E2 -11159.999} C_VEL
LIN {X 0,Y 397.373,Z 208.298,A -85,B 0,C 180,E1 -11163.041,E2 -11163.041} C_VEL
LIN {X 0,Y 397.363,Z 208.3,A -85,B 0,C 180,E1 -11166.091,E2 -11166.091} C_VEL
LIN {X 0,Y 397.236,Z 208.317,A -85,B 0,C 180,E1 -11169.162,E2 -11169.162} C_VEL
LIN {X 0,Y 397.219,Z 208.316,A -85,B 0,C 180,E1 -11172.258,E2 -11172.258} C_VEL
LIN {X 0,Y 397.178,Z 208.322,A -85,B 0,C 180,E1 -11175.392,E2 -11175.392} C_VEL
LIN {X 0,Y 397.158,Z 208.323,A -85,B 0,C 180,E1 -11178.573,E2 -11178.573} C_VEL
LIN {X 0,Y 397.097,Z 208.33,A -85,B 0,C 180,E1 -11181.818,E2 -11181.818} C_VEL
LIN {X 0,Y 397.156,Z 208.323,A -85,B 0,C 180,E1 -11185.131,E2 -11185.131} C_VEL
LIN {X 0,Y 397.163,Z 208.326,A -85,B 0,C 180,E1 -11187.775,E2 -11187.775} C_VEL
LIN {X 0,Y 397.079,Z 208.337,A -85,B 0,C 180,E1 -11190.882,E2 -11190.882} C_VEL
LIN {X 0,Y 397.12,Z 208.327,A -85,B 0,C 180,E1 -11194.493,E2 -11194.493} C_VEL
LIN {X 0,Y 397.101,Z 208.331,A -85,B 0,C 180,E1 -11198.275,E2 -11198.275} C_VEL
LIN {X 0,Y 397.064,Z 208.329,A -85,B 0,C 180,E1 -11200.911,E2 -11200.911} C_VEL
LIN {X 0,Y 397.101,Z 208.333,A -85,B 0,C 180,E1 -11203.648,E2 -11203.648} C_VEL
LIN {X 0,Y 397.099,Z 208.339,A -85,B 0,C 180,E1 -11206.521,E2 -11206.521} C_VEL
LIN {X 0,Y 397.088,Z 208.33,A -85,B 0,C 180,E1 -11210.418,E2 -11210.418} C_VEL
LIN {X 0,Y 397.09,Z 208.44,A -85,B 0,C 180,E1 -11210.976,E2 -11210.976} C_VEL
LIN {X 0,Y 402.504,Z 223.66,A -85,B 0,C 180,E1 -11213.857,E2 -11213.857} C_VEL
LIN {X 0,Y 404.478,Z 229.429,A -85,B 0,C 180,E1 -11214.858,E2 -11214.858} C_VEL
LIN {X 0,Y 414.46,Z 249.081,A -85,B 0,C 180,E1 -11216.307,E2 -11216.307} C_VEL
LIN {X 0,Y 417.126,Z 255.299,A -85,B 0,C 180,E1 -11216.698,E2 -11216.698} C_VEL
LIN {X 0,Y 419.196,Z 268.694,A -85,B 0,C 180,E1 -11217.176,E2 -11217.176} C_VEL
LIN {X 0,Y 414.633,Z 437.854,A -85,B 0,C 180,E1 -11220.303,E2 -11220.303} C_VEL
LIN {X 0,Y 413.552,Z 454.36,A -85,B 0,C 180,E1 -11220.786,E2 -11220.786} C_VEL
LIN {X 0,Y 412.303,Z 469.773,A -85,B 0,C 180,E1 -11221.421,E2 -11221.421} C_VEL
LIN {X 0,Y 410.86,Z 484.75,A -85,B 0,C 180,E1 -11222.215,E2 -11222.215} C_VEL
LIN {X 0,Y 408.995,Z 500.765,A -85,B 0,C 180,E1 -11223.279,E2 -11223.279} C_VEL
LIN {X 0,Y 406.974,Z 516.274,A -85,B 0,C 180,E1 -11224.559,E2 -11224.559} C_VEL
LIN {X 0,Y 405.117,Z 529.993,A -85,B 0,C 180,E1 -11225.939,E2 -11225.939} C_VEL
LIN {X 0,Y 403.564,Z 540.763,A -85,B 0,C 180,E1 -11227.201,E2 -11227.201} C_VEL
LIN {X 0,Y 401.651,Z 553.735,A -85,B 0,C 180,E1 -11228.978,E2 -11228.978} C_VEL
LIN {X 0,Y 400.108,Z 564.727,A -85,B 0,C 180,E1 -11230.769,E2 -11230.769} C_VEL
LIN {X 0,Y 398.874,Z 574.121,A -85,B 0,C 180,E1 -11232.569,E2 -11232.569} C_VEL
LIN {X 0,Y 397.71,Z 583.289,A -85,B 0,C 180,E1 -11234.627,E2 -11234.627} C_VEL
LIN {X 0,Y 396.887,Z 591.621,A -85,B 0,C 180,E1 -11236.886,E2 -11236.886} C_VEL
LIN {X 0,Y 396.227,Z 598.706,A -85,B 0,C 180,E1 -11239.264,E2 -11239.264} C_VEL
LIN {X 0,Y 395.913,Z 604.591,A -85,B 0,C 180,E1 -11241.834,E2 -11241.834} C_VEL
LIN {X 0,Y 395.819,Z 608.03,A -85,B 0,C 180,E1 -11243.882,E2 -11243.882} C_VEL
LIN {X 0,Y 395.725,Z 610.528,A -85,B 0,C 180,E1 -11245.924,E2 -11245.924} C_VEL
LIN {X 0,Y 395.778,Z 611.943,A -85,B 0,C 180,E1 -11247.962,E2 -11247.962} C_VEL
LIN {X 0,Y 395.773,Z 612.465,A -85,B 0,C 180,E1 -11249.998,E2 -11249.998} C_VEL
LIN {X 0,Y 395.793,Z 611.924,A -85,B 0,C 180,E1 -11252.033,E2 -11252.033} C_VEL
LIN {X 0,Y 395.723,Z 610.485,A -85,B 0,C 180,E1 -11254.071,E2 -11254.071} C_VEL
LIN {X 0,Y 395.854,Z 607.891,A -85,B 0,C 180,E1 -11256.164,E2 -11256.164} C_VEL
LIN {X 0,Y 395.909,Z 604.472,A -85,B 0,C 180,E1 -11258.162,E2 -11258.162} C_VEL
LIN {X 0,Y 396.086,Z 599.83,A -85,B 0,C 180,E1 -11260.218,E2 -11260.218} C_VEL
LIN {X 0,Y 396.627,Z 594.044,A -85,B 0,C 180,E1 -11262.274,E2 -11262.274} C_VEL
LIN {X 0,Y 397.242,Z 587.022,A -85,B 0,C 180,E1 -11264.338,E2 -11264.338} C_VEL
LIN {X 0,Y 398.43,Z 577.355,A -85,B 0,C 180,E1 -11266.654,E2 -11266.654} C_VEL
LIN {X 0,Y 399.618,Z 566.95,A -85,B 0,C 180,E1 -11268.718,E2 -11268.718} C_VEL
LIN {X 0,Y 401.124,Z 556.199,A -85,B 0,C 180,E1 -11270.509,E2 -11270.509} C_VEL
LIN {X 0,Y 402.838,Z 543.852,A -85,B 0,C 180,E1 -11272.258,E2 -11272.258} C_VEL
LIN {X 0,Y 404.605,Z 530.853,A -85,B 0,C 180,E1 -11273.816,E2 -11273.816} C_VEL
LIN {X 0,Y 406.43,Z 517.116,A -85,B 0,C 180,E1 -11275.199,E2 -11275.199} C_VEL
LIN {X 0,Y 408.155,Z 503.089,A -85,B 0,C 180,E1 -11276.367,E2 -11276.367} C_VEL
LIN {X 0,Y 409.903,Z 487.504,A -85,B 0,C 180,E1 -11277.434,E2 -11277.434} C_VEL
LIN {X 0,Y 411.443,Z 471.762,A -85,B 0,C 180,E1 -11278.291,E2 -11278.291} C_VEL
LIN {X 0,Y 412.638,Z 455.782,A -85,B 0,C 180,E1 -11278.966,E2 -11278.966} C_VEL
LIN {X 0,Y 413.789,Z 438.412,A -85,B 0,C 180,E1 -11279.469,E2 -11279.469} C_VEL
LIN {X 0,Y 418.005,Z 268.878,A -85,B 0,C 180,E1 -11282.567,E2 -11282.567} C_VEL
LIN {X 0,Y 415.547,Z 253.522,A -85,B 0,C 180,E1 -11283.088,E2 -11283.088} C_VEL
LIN {X 0,Y 404.376,Z 230.23,A -85,B 0,C 180,E1 -11284.577,E2 -11284.577} C_VEL
LIN {X 0,Y 398.979,Z 214.139,A -85,B 0,C 180,E1 -11287.305,E2 -11287.305} C_VEL
LIN {X 0,Y 397.086,Z 208.336,A -85,B 0,C 180,E1 -11288.345,E2 -11288.345} C_VEL
LIN {X 0,Y 397.069,Z 208.336,A -85,B 0,C 180,E1 -11290.906,E2 -11290.906} C_VEL
LIN {X 0,Y 397.08,Z 208.336,A -85,B 0,C 180,E1 -11293.646,E2 -11293.646} C_VEL
LIN {X 0,Y 397.084,Z 208.331,A -85,B 0,C 180,E1 -11296.518,E2 -11296.518} C_VEL
LIN {X 0,Y 397.096,Z 208.326,A -85,B 0,C 180,E1 -11299.549,E2 -11299.549} C_VEL
LIN {X 0,Y 397.073,Z 208.328,A -85,B 0,C 180,E1 -11302.788,E2 -11302.788} C_VEL
LIN {X 0,Y 397.092,Z 208.333,A -85,B 0,C 180,E1 -11306.28,E2 -11306.28} C_VEL
LIN {X 0,Y 397.077,Z 208.334,A -85,B 0,C 180,E1 -11310.134,E2 -11310.134} C_VEL
LIN {X 0,Y 397.165,Z 208.315,A -85,B 0,C 180,E1 -11312.608,E2 -11312.608} C_VEL
LIN {X 0,Y 397.106,Z 208.33,A -85,B 0,C 180,E1 -11315.981,E2 -11315.981} C_VEL
LIN {X 0,Y 397.125,Z 208.312,A -85,B 0,C 180,E1 -11319.272,E2 -11319.272} C_VEL
LIN {X 0,Y 397.151,Z 208.324,A -85,B 0,C 180,E1 -11322.844,E2 -11322.844} C_VEL
LIN {X 0,Y 397.195,Z 208.298,A -85,B 0,C 180,E1 -11326.678,E2 -11326.678} C_VEL
LIN {X 0,Y 397.198,Z 208.311,A -85,B 0,C 180,E1 -11329.809,E2 -11329.809} C_VEL
LIN {X 0,Y 397.325,Z 208.302,A -85,B 0,C 180,E1 -11332.888,E2 -11332.888} C_VEL
LIN {X 0,Y 397.229,Z 208.294,A -85,B 0,C 180,E1 -11334.925,E2 -11334.925} C_VEL
LIN {X 0,Y 397.42,Z 208.274,A -85,B 0,C 180,E1 -11337.974,E2 -11337.974} C_VEL
LIN {X 0,Y 397.549,Z 208.273,A -85,B 0,C 180,E1 -11340.001,E2 -11340.001} C_VEL
LIN {X 0,Y 397.349,Z 208.291,A -85,B 0,C 180,E1 -11343.042,E2 -11343.042} C_VEL
LIN {X 0,Y 397.315,Z 208.299,A -85,B 0,C 180,E1 -11346.696,E2 -11346.696} C_VEL
LIN {X 0,Y 397.222,Z 208.312,A -85,B 0,C 180,E1 -11349.163,E2 -11349.163} C_VEL
LIN {X 0,Y 397.189,Z 208.301,A -85,B 0,C 180,E1 -11352.26,E2 -11352.26} C_VEL
LIN {X 0,Y 397.154,Z 208.322,A -85,B 0,C 180,E1 -11355.394,E2 -11355.394} C_VEL
LIN {X 0,Y 397.133,Z 208.31,A -85,B 0,C 180,E1 -11358.575,E2 -11358.575} C_VEL
LIN {X 0,Y 397.07,Z 208.333,A -85,B 0,C 180,E1 -11361.821,E2 -11361.821} C_VEL
LIN {X 0,Y 397.13,Z 208.313,A -85,B 0,C 180,E1 -11365.134,E2 -11365.134} C_VEL
LIN {X 0,Y 397.136,Z 208.32,A -85,B 0,C 180,E1 -11367.778,E2 -11367.778} C_VEL
LIN {X 0,Y 397.054,Z 208.332,A -85,B 0,C 180,E1 -11370.885,E2 -11370.885} C_VEL
LIN {X 0,Y 397.103,Z 208.327,A -85,B 0,C 180,E1 -11374.496,E2 -11374.496} C_VEL
LIN {X 0,Y 397.078,Z 208.324,A -85,B 0,C 180,E1 -11378.279,E2 -11378.279} C_VEL
LIN {X 0,Y 397.069,Z 208.334,A -85,B 0,C 180,E1 -11380.912,E2 -11380.912} C_VEL
LIN {X 0,Y 397.083,Z 208.333,A -85,B 0,C 180,E1 -11383.652,E2 -11383.652} C_VEL
LIN {X 0,Y 397.084,Z 208.331,A -85,B 0,C 180,E1 -11386.525,E2 -11386.525} C_VEL
LIN {X 0,Y 397.077,Z 208.325,A -85,B 0,C 180,E1 -11390.423,E2 -11390.423} C_VEL
LIN {X 0,Y 397.088,Z 208.333,A -85,B 0,C 180,E1 -11393.009,E2 -11393.009} C_VEL
LIN {X 0,Y 397.108,Z 208.325,A -85,B 0,C 180,E1 -11396.286,E2 -11396.286} C_VEL
LIN {X 0,Y 397.091,Z 208.326,A -85,B 0,C 180,E1 -11400.14,E2 -11400.14} C_VEL
LIN {X 0,Y 397.088,Z 208.329,A -85,B 0,C 180,E1 -11403.742,E2 -11403.742} C_VEL
LIN {X 0,Y 397.098,Z 208.329,A -85,B 0,C 180,E1 -11407.089,E2 -11407.089} C_VEL
LIN {X 0,Y 397.142,Z 208.323,A -85,B 0,C 180,E1 -11410.356,E2 -11410.356} C_VEL
LIN {X 0,Y 397.126,Z 208.327,A -85,B 0,C 180,E1 -11413.555,E2 -11413.555} C_VEL
LIN {X 0,Y 397.229,Z 208.317,A -85,B 0,C 180,E1 -11416.706,E2 -11416.706} C_VEL
LIN {X 0,Y 397.215,Z 208.318,A -85,B 0,C 180,E1 -11419.812,E2 -11419.812} C_VEL
LIN {X 0,Y 397.248,Z 208.317,A -85,B 0,C 180,E1 -11421.425,E2 -11421.425} C_VEL
LIN {X 0,Y 398.216,Z 211.168,A -85,B 0,C 180,E1 -11421.923,E2 -11421.923} C_VEL
LIN {X 0,Y 406.928,Z 227.614,A -85,B 0,C 180,E1 -11423.095,E2 -11423.095} C_VEL
LIN {X 0,Y 416.567,Z 247.139,A -85,B 0,C 180,E1 -11424.353,E2 -11424.353} C_VEL
LIN {X 0,Y 418.248,Z 250.924,A -85,B 0,C 180,E1 -11424.572,E2 -11424.572} C_VEL
LIN {X 0,Y 414.274,Z 409.623,A -85,B 0,C 180,E1 -11427.446,E2 -11427.446} C_VEL
LIN {X 0,Y 413.484,Z 415.447,A -85,B 0,C 180,E1 -11427.521,E2 -11427.521} C_VEL
LIN {X 0,Y 407.994,Z 432.4,A -85,B 0,C 180,E1 -11427.663,E2 -11427.663} C_VEL
LIN {X 0,Y 406.635,Z 438.072,A -85,B 0,C 180,E1 -11427.8,E2 -11427.8} C_VEL
LIN {X 0,Y 406.445,Z 439.966,A -85,B 0,C 180,E1 -11427.874,E2 -11427.874} C_VEL
LIN {X 0,Y 405.155,Z 456.079,A -85,B 0,C 180,E1 -11428.636,E2 -11428.636} C_VEL
LIN {X 0,Y 403.759,Z 470.549,A -85,B 0,C 180,E1 -11429.504,E2 -11429.504} C_VEL
LIN {X 0,Y 402.038,Z 485.618,A -85,B 0,C 180,E1 -11430.628,E2 -11430.628} C_VEL
LIN {X 0,Y 400.225,Z 499.634,A -85,B 0,C 180,E1 -11431.894,E2 -11431.894} C_VEL
LIN {X 0,Y 398.285,Z 513.683,A -85,B 0,C 180,E1 -11433.417,E2 -11433.417} C_VEL
LIN {X 0,Y 396.695,Z 524.79,A -85,B 0,C 180,E1 -11434.83,E2 -11434.83} C_VEL
LIN {X 0,Y 394.869,Z 536.851,A -85,B 0,C 180,E1 -11436.646,E2 -11436.646} C_VEL
LIN {X 0,Y 393.344,Z 547.126,A -85,B 0,C 180,E1 -11438.479,E2 -11438.479} C_VEL
LIN {X 0,Y 391.889,Z 557.14,A -85,B 0,C 180,E1 -11440.594,E2 -11440.594} C_VEL
LIN {X 0,Y 390.927,Z 564.613,A -85,B 0,C 180,E1 -11442.461,E2 -11442.461} C_VEL
LIN {X 0,Y 390.086,Z 571.723,A -85,B 0,C 180,E1 -11444.612,E2 -11444.612} C_VEL
LIN {X 0,Y 389.385,Z 577.971,A -85,B 0,C 180,E1 -11446.941,E2 -11446.941} C_VEL
LIN {X 0,Y 389.041,Z 582.324,A -85,B 0,C 180,E1 -11448.978,E2 -11448.978} C_VEL
LIN {X 0,Y 388.683,Z 585.842,A -85,B 0,C 180,E1 -11451.202,E2 -11451.202} C_VEL
LIN {X 0,Y 388.457,Z 588.269,A -85,B 0,C 180,E1 -11453.457,E2 -11453.457} C_VEL
LIN {X 0,Y 388.412,Z 589.607,A -85,B 0,C 180,E1 -11455.74,E2 -11455.74} C_VEL
LIN {X 0,Y 388.452,Z 589.703,A -85,B 0,C 180,E1 -11458.062,E2 -11458.062} C_VEL
LIN {X 0,Y 388.522,Z 588.61,A -85,B 0,C 180,E1 -11460.432,E2 -11460.432} C_VEL
LIN {X 0,Y 388.716,Z 586.233,A -85,B 0,C 180,E1 -11462.849,E2 -11462.849} C_VEL
LIN {X 0,Y 389.069,Z 582.42,A -85,B 0,C 180,E1 -11465.314,E2 -11465.314} C_VEL
LIN {X 0,Y 389.663,Z 576.983,A -85,B 0,C 180,E1 -11467.825,E2 -11467.825} C_VEL
LIN {X 0,Y 390.233,Z 571.665,A -85,B 0,C 180,E1 -11469.76,E2 -11469.76} C_VEL
LIN {X 0,Y 391.255,Z 563.678,A -85,B 0,C 180,E1 -11472.145,E2 -11472.145} C_VEL
LIN {X 0,Y 392.533,Z 554.918,A -85,B 0,C 180,E1 -11474.289,E2 -11474.289} C_VEL
LIN {X 0,Y 394.172,Z 544.789,A -85,B 0,C 180,E1 -11476.345,E2 -11476.345} C_VEL
LIN {X 0,Y 395.832,Z 533.8,A -85,B 0,C 180,E1 -11478.221,E2 -11478.221} C_VEL
LIN {X 0,Y 397.63,Z 522.488,A -85,B 0,C 180,E1 -11479.858,E2 -11479.858} C_VEL
LIN {X 0,Y 399.476,Z 510.652,A -85,B 0,C 180,E1 -11481.325,E2 -11481.325} C_VEL
LIN {X 0,Y 401.488,Z 496.555,A -85,B 0,C 180,E1 -11482.795,E2 -11482.795} C_VEL
LIN {X 0,Y 403.495,Z 481.217,A -85,B 0,C 180,E1 -11484.11,E2 -11484.11} C_VEL
LIN {X 0,Y 405.155,Z 466.544,A -85,B 0,C 180,E1 -11485.136,E2 -11485.136} C_VEL
LIN {X 0,Y 406.73,Z 450.373,A -85,B 0,C 180,E1 -11486.039,E2 -11486.039} C_VEL
LIN {X 0,Y 407.952,Z 435.049,A -85,B 0,C 180,E1 -11486.696,E2 -11486.696} C_VEL
LIN {X 0,Y 408.889,Z 418.559,A -85,B 0,C 180,E1 -11487.206,E2 -11487.206} C_VEL
LIN {X 0,Y 410.569,Z 358.901,A -85,B 0,C 180,E1 -11488.348,E2 -11488.348} C_VEL
LIN {X 0,Y 413.551,Z 253.71,A -85,B 0,C 180,E1 -11490.319,E2 -11490.319} C_VEL
LIN {X 0,Y 404.474,Z 235.527,A -85,B 0,C 180,E1 -11491.641,E2 -11491.641} C_VEL
LIN {X 0,Y 394.857,Z 218.537,A -85,B 0,C 180,E1 -11493.1,E2 -11493.1} C_VEL
LIN {X 0,Y 391.138,Z 212.322,A -85,B 0,C 180,E1 -11493.697,E2 -11493.697} C_VEL
LIN {X 0,Y 390.12,Z 209.202,A -85,B 0,C 180,E1 -11494.382,E2 -11494.382} C_VEL
LIN {X 0,Y 390.041,Z 209.219,A -85,B 0,C 180,E1 -11497.765,E2 -11497.765} C_VEL
LIN {X 0,Y 390.108,Z 209.206,A -85,B 0,C 180,E1 -11501.077,E2 -11501.077} C_VEL
LIN {X 0,Y 390.141,Z 209.201,A -85,B 0,C 180,E1 -11504.323,E2 -11504.323} C_VEL
LIN {X 0,Y 390.172,Z 209.194,A -85,B 0,C 180,E1 -11507.516,E2 -11507.516} C_VEL
LIN {X 0,Y 390.206,Z 209.191,A -85,B 0,C 180,E1 -11510.671,E2 -11510.671} C_VEL
LIN {X 0,Y 390.327,Z 209.175,A -85,B 0,C 180,E1 -11513.798,E2 -11513.798} C_VEL
LIN {X 0,Y 390.417,Z 209.166,A -85,B 0,C 180,E1 -11517.936,E2 -11517.936} C_VEL
LIN {X 0,Y 390.548,Z 209.151,A -85,B 0,C 180,E1 -11519.999,E2 -11519.999} C_VEL
LIN {X 0,Y 390.308,Z 209.179,A -85,B 0,C 180,E1 -11523.096,E2 -11523.096} C_VEL
LIN {X 0,Y 390.316,Z 209.177,A -85,B 0,C 180,E1 -11526.202,E2 -11526.202} C_VEL
LIN {X 0,Y 390.194,Z 209.195,A -85,B 0,C 180,E1 -11529.329,E2 -11529.329} C_VEL
LIN {X 0,Y 390.171,Z 209.193,A -85,B 0,C 180,E1 -11532.483,E2 -11532.483} C_VEL
LIN {X 0,Y 390.139,Z 209.196,A -85,B 0,C 180,E1 -11535.676,E2 -11535.676} C_VEL
LIN {X 0,Y 390.102,Z 209.201,A -85,B 0,C 180,E1 -11538.922,E2 -11538.922} C_VEL
LIN {X 0,Y 390.04,Z 209.209,A -85,B 0,C 180,E1 -11542.234,E2 -11542.234} C_VEL
LIN {X 0,Y 390.12,Z 209.203,A -85,B 0,C 180,E1 -11545.742,E2 -11545.742} C_VEL
LIN {X 0,Y 390.054,Z 209.21,A -85,B 0,C 180,E1 -11549.109,E2 -11549.109} C_VEL
LIN {X 0,Y 390.042,Z 209.21,A -85,B 0,C 180,E1 -11552.721,E2 -11552.721} C_VEL
LIN {X 0,Y 390.055,Z 209.209,A -85,B 0,C 180,E1 -11555.824,E2 -11555.824} C_VEL
LIN {X 0,Y 390.069,Z 209.211,A -85,B 0,C 180,E1 -11559.217,E2 -11559.217} C_VEL
LIN {X 0,Y 390.057,Z 209.214,A -85,B 0,C 180,E1 -11563.21,E2 -11563.21} C_VEL
LIN {X 0,Y 390.053,Z 209.212,A -85,B 0,C 180,E1 -11566.788,E2 -11566.788} C_VEL
LIN {X 0,Y 390.057,Z 209.336,A -85,B 0,C 180,E1 -11570.236,E2 -11570.236} C_VEL
LIN {X 0,Y 395.377,Z 223.954,A -85,B 0,C 180,E1 -11573.119,E2 -11573.119} C_VEL
LIN {X 0,Y 397.156,Z 229.22,A -85,B 0,C 180,E1 -11574.053,E2 -11574.053} C_VEL
LIN {X 0,Y 404.562,Z 243.305,A -85,B 0,C 180,E1 -11575.182,E2 -11575.182} C_VEL
LIN {X 0,Y 411.456,Z 257.581,A -85,B 0,C 180,E1 -11576.197,E2 -11576.197} C_VEL
LIN {X 0,Y 413.304,Z 269.863,A -85,B 0,C 180,E1 -11576.644,E2 -11576.644} C_VEL
LIN {X 0,Y 408.548,Z 437.779,A -85,B 0,C 180,E1 -11579.797,E2 -11579.797} C_VEL
LIN {X 0,Y 407.392,Z 454.702,A -85,B 0,C 180,E1 -11580.3,E2 -11580.3} C_VEL
LIN {X 0,Y 406.088,Z 469.952,A -85,B 0,C 180,E1 -11580.942,E2 -11580.942} C_VEL
LIN {X 0,Y 404.336,Z 486.8,A -85,B 0,C 180,E1 -11581.868,E2 -11581.868} C_VEL
LIN {X 0,Y 402.393,Z 502.558,A -85,B 0,C 180,E1 -11582.966,E2 -11582.966} C_VEL
LIN {X 0,Y 400.336,Z 517.516,A -85,B 0,C 180,E1 -11584.245,E2 -11584.245} C_VEL
LIN {X 0,Y 398.411,Z 531.084,A -85,B 0,C 180,E1 -11585.647,E2 -11585.647} C_VEL
LIN {X 0,Y 396.662,Z 542.618,A -85,B 0,C 180,E1 -11587.057,E2 -11587.057} C_VEL
LIN {X 0,Y 394.683,Z 555.251,A -85,B 0,C 180,E1 -11588.862,E2 -11588.862} C_VEL
LIN {X 0,Y 393.081,Z 566.033,A -85,B 0,C 180,E1 -11590.683,E2 -11590.683} C_VEL
LIN {X 0,Y 391.676,Z 576.463,A -85,B 0,C 180,E1 -11592.777,E2 -11592.777} C_VEL
LIN {X 0,Y 390.509,Z 585.164,A -85,B 0,C 180,E1 -11594.871,E2 -11594.871} C_VEL
LIN {X 0,Y 389.764,Z 592.498,A -85,B 0,C 180,E1 -11596.984,E2 -11596.984} C_VEL
LIN {X 0,Y 389.194,Z 598.524,A -85,B 0,C 180,E1 -11599.068,E2 -11599.068} C_VEL
LIN {X 0,Y 388.841,Z 604.404,A -85,B 0,C 180,E1 -11601.684,E2 -11601.684} C_VEL
LIN {X 0,Y 388.723,Z 608.054,A -85,B 0,C 180,E1 -11603.92,E2 -11603.92} C_VEL
LIN {X 0,Y 388.648,Z 610.332,A -85,B 0,C 180,E1 -11605.85,E2 -11605.85} C_VEL
LIN {X 0,Y 388.675,Z 611.742,A -85,B 0,C 180,E1 -11607.925,E2 -11607.925} C_VEL
LIN {X 0,Y 388.703,Z 612.258,A -85,B 0,C 180,E1 -11609.998,E2 -11609.998} C_VEL
LIN {X 0,Y 388.689,Z 611.712,A -85,B 0,C 180,E1 -11612.07,E2 -11612.07} C_VEL
LIN {X 0,Y 388.647,Z 610.264,A -85,B 0,C 180,E1 -11614.145,E2 -11614.145} C_VEL
LIN {X 0,Y 388.753,Z 607.738,A -85,B 0,C 180,E1 -11616.224,E2 -11616.224} C_VEL
LIN {X 0,Y 388.838,Z 604.233,A -85,B 0,C 180,E1 -11618.311,E2 -11618.311} C_VEL
LIN {X 0,Y 389.031,Z 599.583,A -85,B 0,C 180,E1 -11620.405,E2 -11620.405} C_VEL
LIN {X 0,Y 389.617,Z 593.784,A -85,B 0,C 180,E1 -11622.498,E2 -11622.498} C_VEL
LIN {X 0,Y 390.255,Z 586.749,A -85,B 0,C 180,E1 -11624.6,E2 -11624.6} C_VEL
LIN {X 0,Y 391.517,Z 577.066,A -85,B 0,C 180,E1 -11626.956,E2 -11626.956} C_VEL
LIN {X 0,Y 392.79,Z 566.645,A -85,B 0,C 180,E1 -11629.055,E2 -11629.055} C_VEL
LIN {X 0,Y 394.353,Z 555.87,A -85,B 0,C 180,E1 -11630.878,E2 -11630.878} C_VEL
LIN {X 0,Y 396.045,Z 544.367,A -85,B 0,C 180,E1 -11632.54,E2 -11632.54} C_VEL
LIN {X 0,Y 397.857,Z 531.639,A -85,B 0,C 180,E1 -11634.107,E2 -11634.107} C_VEL
LIN {X 0,Y 399.741,Z 517.993,A -85,B 0,C 180,E1 -11635.511,E2 -11635.511} C_VEL
LIN {X 0,Y 401.573,Z 503.732,A -85,B 0,C 180,E1 -11636.733,E2 -11636.733} C_VEL
LIN {X 0,Y 403.356,Z 488.907,A -85,B 0,C 180,E1 -11637.777,E2 -11637.777} C_VEL
LIN {X 0,Y 404.919,Z 473.646,A -85,B 0,C 180,E1 -11638.647,E2 -11638.647} C_VEL
LIN {X 0,Y 406.279,Z 456.658,A -85,B 0,C 180,E1 -11639.392,E2 -11639.392} C_VEL
LIN {X 0,Y 407.444,Z 439.624,A -85,B 0,C 180,E1 -11639.904,E2 -11639.904} C_VEL
LIN {X 0,Y 408.261,Z 410.805,A -85,B 0,C 180,E1 -11640.47,E2 -11640.47} C_VEL
LIN {X 0,Y 411.903,Z 269.074,A -85,B 0,C 180,E1 -11643.078,E2 -11643.078} C_VEL
LIN {X 0,Y 409.713,Z 256.254,A -85,B 0,C 180,E1 -11643.536,E2 -11643.536} C_VEL
LIN {X 0,Y 398.958,Z 233.873,A -85,B 0,C 180,E1 -11644.996,E2 -11644.996} C_VEL
LIN {X 0,Y 396.992,Z 229.835,A -85,B 0,C 180,E1 -11645.302,E2 -11645.302} C_VEL
LIN {X 0,Y 391.38,Z 213.196,A -85,B 0,C 180,E1 -11648.213,E2 -11648.213} C_VEL
LIN {X 0,Y 390.085,Z 209.209,A -85,B 0,C 180,E1 -11648.939,E2 -11648.939} C_VEL
LIN {X 0,Y 390.021,Z 209.208,A -85,B 0,C 180,E1 -11652.371,E2 -11652.371} C_VEL
LIN {X 0,Y 390.024,Z 209.207,A -85,B 0,C 180,E1 -11655.352,E2 -11655.352} C_VEL
LIN {X 0,Y 390.046,Z 209.211,A -85,B 0,C 180,E1 -11658.189,E2 -11658.189} C_VEL
LIN {X 0,Y 390.07,Z 209.209,A -85,B 0,C 180,E1 -11660.906,E2 -11660.906} C_VEL
LIN {X 0,Y 390.059,Z 209.205,A -85,B 0,C 180,E1 -11664.791,E2 -11664.791} C_VEL
LIN {X 0,Y 389.995,Z 209.201,A -85,B 0,C 180,E1 -11668.494,E2 -11668.494} C_VEL
LIN {X 0,Y 390.089,Z 209.203,A -85,B 0,C 180,E1 -11672.068,E2 -11672.068} C_VEL
LIN {X 0,Y 390.053,Z 209.21,A -85,B 0,C 180,E1 -11675.518,E2 -11675.518} C_VEL
LIN {X 0,Y 390.073,Z 209.194,A -85,B 0,C 180,E1 -11678.879,E2 -11678.879} C_VEL
LIN {X 0,Y 390.1,Z 209.196,A -85,B 0,C 180,E1 -11682.166,E2 -11682.166} C_VEL
LIN {X 0,Y 390.116,Z 209.195,A -85,B 0,C 180,E1 -11685.392,E2 -11685.392} C_VEL
LIN {X 0,Y 390.128,Z 209.173,A -85,B 0,C 180,E1 -11688.571,E2 -11688.571} C_VEL
LIN {X 0,Y 390.277,Z 209.181,A -85,B 0,C 180,E1 -11692.031,E2 -11692.031} C_VEL
LIN {X 0,Y 390.201,Z 209.17,A -85,B 0,C 180,E1 -11694.834,E2 -11694.834} C_VEL
LIN {X 0,Y 390.389,Z 209.149,A -85,B 0,C 180,E1 -11697.937,E2 -11697.937} C_VEL
LIN {X 0,Y 390.519,Z 209.148,A -85,B 0,C 180,E1 -11700.001,E2 -11700.001} C_VEL
LIN {X 0,Y 390.284,Z 209.17,A -85,B 0,C 180,E1 -11703.097,E2 -11703.097} C_VEL
LIN {X 0,Y 390.269,Z 209.175,A -85,B 0,C 180,E1 -11706.692,E2 -11706.692} C_VEL
LIN {X 0,Y 390.174,Z 209.189,A -85,B 0,C 180,E1 -11709.33,E2 -11709.33} C_VEL
LIN {X 0,Y 390.165,Z 209.188,A -85,B 0,C 180,E1 -11713.44,E2 -11713.44} C_VEL
LIN {X 0,Y 390.122,Z 209.191,A -85,B 0,C 180,E1 -11717.31,E2 -11717.31} C_VEL
LIN {X 0,Y 390.06,Z 209.199,A -85,B 0,C 180,E1 -11720.472,E2 -11720.472} C_VEL
LIN {X 0,Y 390.063,Z 209.205,A -85,B 0,C 180,E1 -11723.353,E2 -11723.353} C_VEL
LIN {X 0,Y 390.088,Z 209.192,A -85,B 0,C 180,E1 -11726.771,E2 -11726.771} C_VEL
LIN {X 0,Y 390.015,Z 209.216,A -85,B 0,C 180,E1 -11730.303,E2 -11730.303} C_VEL
LIN {X 0,Y 390.046,Z 209.199,A -85,B 0,C 180,E1 -11734.027,E2 -11734.027} C_VEL
LIN {X 0,Y 390.021,Z 209.211,A -85,B 0,C 180,E1 -11737.553,E2 -11737.553} C_VEL
LIN {X 0,Y 390.037,Z 209.21,A -85,B 0,C 180,E1 -11740.824,E2 -11740.824} C_VEL
LIN {X 0,Y 390.037,Z 209.208,A -85,B 0,C 180,E1 -11743.889,E2 -11743.889} C_VEL
LIN {X 0,Y 390.039,Z 209.211,A -85,B 0,C 180,E1 -11746.793,E2 -11746.793} C_VEL
LIN {X 0,Y 390.041,Z 209.208,A -85,B 0,C 180,E1 -11749.564,E2 -11749.564} C_VEL
LIN {X 0,Y 390.03,Z 209.215,A -85,B 0,C 180,E1 -11752.453,E2 -11752.453} C_VEL
LIN {X 0,Y 390.058,Z 209.2,A -85,B 0,C 180,E1 -11755.979,E2 -11755.979} C_VEL
LIN {X 0,Y 390.028,Z 209.207,A -85,B 0,C 180,E1 -11759.704,E2 -11759.704} C_VEL
LIN {X 0,Y 390.048,Z 209.209,A -85,B 0,C 180,E1 -11763.231,E2 -11763.231} C_VEL
LIN {X 0,Y 390.062,Z 209.206,A -85,B 0,C 180,E1 -11766.767,E2 -11766.767} C_VEL
LIN {X 0,Y 390.1,Z 209.204,A -85,B 0,C 180,E1 -11769.986,E2 -11769.986} C_VEL
LIN {X 0,Y 390.104,Z 209.203,A -85,B 0,C 180,E1 -11773.25,E2 -11773.25} C_VEL
LIN {X 0,Y 390.195,Z 209.192,A -85,B 0,C 180,E1 -11776.565,E2 -11776.565} C_VEL
LIN {X 0,Y 390.167,Z 209.197,A -85,B 0,C 180,E1 -11779.626,E2 -11779.626} C_VEL
LIN {X 0,Y 390.218,Z 209.253,A -85,B 0,C 180,E1 -11780.838,E2 -11780.838} C_VEL
LIN {X 0,Y 390.824,Z 211.376,A -85,B 0,C 180,E1 -11781.199,E2 -11781.199} C_VEL
LIN {X 0,Y 400.744,Z 229.44,A -85,B 0,C 180,E1 -11782.563,E2 -11782.563} C_VEL
LIN {X 0,Y 411.555,Z 251.619,A -85,B 0,C 180,E1 -11784.014,E2 -11784.014} C_VEL
LIN {X 0,Y 412.121,Z 253.329,A -85,B 0,C 180,E1 -11784.099,E2 -11784.099} C_VEL
LIN {X 0,Y 407.787,Z 417.165,A -85,B 0,C 180,E1 -11787.131,E2 -11787.131} C_VEL
LIN {X 0,Y 406.859,Z 434.26,A -85,B 0,C 180,E1 -11787.651,E2 -11787.651} C_VEL
LIN {X 0,Y 406.445,Z 439.966,A -85,B 0,C 180,E1 -11787.874,E2 -11787.874} C_VEL
LIN {X 0,Y 405.379,Z 445.741,A -85,B 0,C 180,E1 -11788.071,E2 -11788.071} C_VEL
LIN {X 0,Y 399.276,Z 462.223,A -85,B 0,C 180,E1 -11788.584,E2 -11788.584} C_VEL
LIN {X 0,Y 397.808,Z 467.465,A -85,B 0,C 180,E1 -11788.847,E2 -11788.847} C_VEL
LIN {X 0,Y 397.543,Z 469.211,A -85,B 0,C 180,E1 -11788.954,E2 -11788.954} C_VEL
LIN {X 0,Y 395.901,Z 483.448,A -85,B 0,C 180,E1 -11790.002,E2 -11790.002} C_VEL
LIN {X 0,Y 394.048,Z 497.453,A -85,B 0,C 180,E1 -11791.24,E2 -11791.24} C_VEL
LIN {X 0,Y 392.073,Z 511.232,A -85,B 0,C 180,E1 -11792.699,E2 -11792.699} C_VEL
LIN {X 0,Y 390.102,Z 524.519,A -85,B 0,C 180,E1 -11794.394,E2 -11794.394} C_VEL
LIN {X 0,Y 388.478,Z 534.818,A -85,B 0,C 180,E1 -11795.942,E2 -11795.942} C_VEL
LIN {X 0,Y 386.768,Z 545.648,A -85,B 0,C 180,E1 -11797.835,E2 -11797.835} C_VEL
LIN {X 0,Y 385.248,Z 555.588,A -85,B 0,C 180,E1 -11799.896,E2 -11799.896} C_VEL
LIN {X 0,Y 384.003,Z 564.596,A -85,B 0,C 180,E1 -11802.152,E2 -11802.152} C_VEL
LIN {X 0,Y 383.107,Z 571.746,A -85,B 0,C 180,E1 -11804.341,E2 -11804.341} C_VEL
LIN {X 0,Y 382.41,Z 577.611,A -85,B 0,C 180,E1 -11806.531,E2 -11806.531} C_VEL
LIN {X 0,Y 381.979,Z 582.419,A -85,B 0,C 180,E1 -11808.785,E2 -11808.785} C_VEL
LIN {X 0,Y 381.688,Z 585.179,A -85,B 0,C 180,E1 -11810.48,E2 -11810.48} C_VEL
LIN {X 0,Y 381.411,Z 588.058,A -85,B 0,C 180,E1 -11812.879,E2 -11812.879} C_VEL
LIN {X 0,Y 381.326,Z 589.681,A -85,B 0,C 180,E1 -11815.431,E2 -11815.431} C_VEL
LIN {X 0,Y 381.378,Z 589.949,A -85,B 0,C 180,E1 -11817.804,E2 -11817.804} C_VEL
LIN {X 0,Y 381.429,Z 589.191,A -85,B 0,C 180,E1 -11820.002,E2 -11820.002} C_VEL
LIN {X 0,Y 381.558,Z 587.221,A -85,B 0,C 180,E1 -11822.288,E2 -11822.288} C_VEL
LIN {X 0,Y 381.864,Z 583.785,A -85,B 0,C 180,E1 -11824.789,E2 -11824.789} C_VEL
LIN {X 0,Y 382.286,Z 580.248,A -85,B 0,C 180,E1 -11826.691,E2 -11826.691} C_VEL
LIN {X 0,Y 382.971,Z 574.417,A -85,B 0,C 180,E1 -11829.115,E2 -11829.115} C_VEL
LIN {X 0,Y 383.852,Z 567.682,A -85,B 0,C 180,E1 -11831.35,E2 -11831.35} C_VEL
LIN {X 0,Y 384.926,Z 560.159,A -85,B 0,C 180,E1 -11833.424,E2 -11833.424} C_VEL
LIN {X 0,Y 386.467,Z 550.867,A -85,B 0,C 180,E1 -11835.544,E2 -11835.544} C_VEL
LIN {X 0,Y 388.164,Z 540.393,A -85,B 0,C 180,E1 -11837.546,E2 -11837.546} C_VEL
LIN {X 0,Y 389.876,Z 530.17,A -85,B 0,C 180,E1 -11839.211,E2 -11839.211} C_VEL
LIN {X 0,Y 391.797,Z 518.465,A -85,B 0,C 180,E1 -11840.848,E2 -11840.848} C_VEL
LIN {X 0,Y 393.946,Z 504.785,A -85,B 0,C 180,E1 -11842.448,E2 -11842.448} C_VEL
LIN {X 0,Y 396.007,Z 490.342,A -85,B 0,C 180,E1 -11843.853,E2 -11843.853} C_VEL
LIN {X 0,Y 397.875,Z 476.025,A -85,B 0,C 180,E1 -11845.002,E2 -11845.002} C_VEL
LIN {X 0,Y 399.612,Z 461.156,A -85,B 0,C 180,E1 -11845.976,E2 -11845.976} C_VEL
LIN {X 0,Y 401.114,Z 444.996,A -85,B 0,C 180,E1 -11846.816,E2 -11846.816} C_VEL
LIN {X 0,Y 402.334,Z 427.983,A -85,B 0,C 180,E1 -11847.468,E2 -11847.468} C_VEL
LIN {X 0,Y 403.133,Z 411.441,A -85,B 0,C 180,E1 -11847.893,E2 -11847.893} C_VEL
LIN {X 0,Y 407.74,Z 256.088,A -85,B 0,C 180,E1 -11850.844,E2 -11850.844} C_VEL
LIN {X 0,Y 398.991,Z 238.62,A -85,B 0,C 180,E1 -11852.162,E2 -11852.162} C_VEL
LIN {X 0,Y 389.948,Z 222.563,A -85,B 0,C 180,E1 -11853.58,E2 -11853.58} C_VEL
LIN {X 0,Y 383.88,Z 212.613,A -85,B 0,C 180,E1 -11854.59,E2 -11854.59} C_VEL
LIN {X 0,Y 383.031,Z 210.09,A -85,B 0,C 180,E1 -11855.183,E2 -11855.183} C_VEL
LIN {X 0,Y 382.996,Z 210.087,A -85,B 0,C 180,E1 -11858.469,E2 -11858.469} C_VEL
LIN {X 0,Y 383.066,Z 210.074,A -85,B 0,C 180,E1 -11861.826,E2 -11861.826} C_VEL
LIN {X 0,Y 383.112,Z 210.073,A -85,B 0,C 180,E1 -11865.118,E2 -11865.118} C_VEL
LIN {X 0,Y 383.098,Z 210.078,A -85,B 0,C 180,E1 -11868.357,E2 -11868.357} C_VEL
LIN {X 0,Y 383.266,Z 210.055,A -85,B 0,C 180,E1 -11871.976,E2 -11871.976} C_VEL
LIN {X 0,Y 383.197,Z 210.064,A -85,B 0,C 180,E1 -11874.738,E2 -11874.738} C_VEL
LIN {X 0,Y 383.385,Z 210.043,A -85,B 0,C 180,E1 -11877.898,E2 -11877.898} C_VEL
LIN {X 0,Y 383.518,Z 210.027,A -85,B 0,C 180,E1 -11879.999,E2 -11879.999} C_VEL
LIN {X 0,Y 383.244,Z 210.059,A -85,B 0,C 180,E1 -11883.153,E2 -11883.153} C_VEL
LIN {X 0,Y 383.271,Z 210.054,A -85,B 0,C 180,E1 -11886.316,E2 -11886.316} C_VEL
LIN {X 0,Y 383.144,Z 210.07,A -85,B 0,C 180,E1 -11889.502,E2 -11889.502} C_VEL
LIN {X 0,Y 383.127,Z 210.07,A -85,B 0,C 180,E1 -11893.535,E2 -11893.535} C_VEL
LIN {X 0,Y 383.095,Z 210.076,A -85,B 0,C 180,E1 -11897.069,E2 -11897.069} C_VEL
LIN {X 0,Y 383.03,Z 210.085,A -85,B 0,C 180,E1 -11900.646,E2 -11900.646} C_VEL
LIN {X 0,Y 383.027,Z 210.082,A -85,B 0,C 180,E1 -11903.807,E2 -11903.807} C_VEL
LIN {X 0,Y 383.081,Z 210.078,A -85,B 0,C 180,E1 -11906.123,E2 -11906.123} C_VEL
LIN {X 0,Y 382.99,Z 210.088,A -85,B 0,C 180,E1 -11909.699,E2 -11909.699} C_VEL
LIN {X 0,Y 383,Z 210.09,A -85,B 0,C 180,E1 -11913.4,E2 -11913.4} C_VEL
LIN {X 0,Y 383.031,Z 210.083,A -85,B 0,C 180,E1 -11916.163,E2 -11916.163} C_VEL
LIN {X 0,Y 382.997,Z 210.089,A -85,B 0,C 180,E1 -11919.959,E2 -11919.959} C_VEL
LIN {X 0,Y 383.008,Z 210.09,A -85,B 0,C 180,E1 -11922.778,E2 -11922.778} C_VEL
LIN {X 0,Y 382.996,Z 210.092,A -85,B 0,C 180,E1 -11925.788,E2 -11925.788} C_VEL
LIN {X 0,Y 382.964,Z 210.097,A -85,B 0,C 180,E1 -11928.799,E2 -11928.799} C_VEL
LIN {X 0,Y 382.987,Z 210.199,A -85,B 0,C 180,E1 -11929.444,E2 -11929.444} C_VEL
LIN {X 0,Y 388.097,Z 224.084,A -85,B 0,C 180,E1 -11932.3,E2 -11932.3} C_VEL
LIN {X 0,Y 389.833,Z 228.913,A -85,B 0,C 180,E1 -11933.199,E2 -11933.199} C_VEL
LIN {X 0,Y 398.525,Z 245.187,A -85,B 0,C 180,E1 -11934.577,E2 -11934.577} C_VEL
LIN {X 0,Y 405.87,Z 260.393,A -85,B 0,C 180,E1 -11935.7,E2 -11935.7} C_VEL
LIN {X 0,Y 407.448,Z 271.461,A -85,B 0,C 180,E1 -11936.104,E2 -11936.104} C_VEL
LIN {X 0,Y 402.546,Z 436.93,A -85,B 0,C 180,E1 -11939.258,E2 -11939.258} C_VEL
LIN {X 0,Y 401.374,Z 453.235,A -85,B 0,C 180,E1 -11939.737,E2 -11939.737} C_VEL
LIN {X 0,Y 400.032,Z 468.837,A -85,B 0,C 180,E1 -11940.387,E2 -11940.387} C_VEL
LIN {X 0,Y 398.344,Z 484.902,A -85,B 0,C 180,E1 -11941.263,E2 -11941.263} C_VEL
LIN {X 0,Y 396.472,Z 499.691,A -85,B 0,C 180,E1 -11942.268,E2 -11942.268} C_VEL
LIN {X 0,Y 394.331,Z 514.793,A -85,B 0,C 180,E1 -11943.539,E2 -11943.539} C_VEL
LIN {X 0,Y 392.22,Z 528.671,A -85,B 0,C 180,E1 -11944.954,E2 -11944.954} C_VEL
LIN {X 0,Y 390.305,Z 540.557,A -85,B 0,C 180,E1 -11946.38,E2 -11946.38} C_VEL
LIN {X 0,Y 388.534,Z 551.775,A -85,B 0,C 180,E1 -11947.953,E2 -11947.953} C_VEL
LIN {X 0,Y 386.73,Z 562.965,A -85,B 0,C 180,E1 -11949.799,E2 -11949.799} C_VEL
LIN {X 0,Y 385.374,Z 571.832,A -85,B 0,C 180,E1 -11951.497,E2 -11951.497} C_VEL
LIN {X 0,Y 384.152,Z 580.858,A -85,B 0,C 180,E1 -11953.525,E2 -11953.525} C_VEL
LIN {X 0,Y 383.096,Z 588.814,A -85,B 0,C 180,E1 -11955.659,E2 -11955.659} C_VEL
LIN {X 0,Y 382.42,Z 595.462,A -85,B 0,C 180,E1 -11957.797,E2 -11957.797} C_VEL
LIN {X 0,Y 381.887,Z 600.875,A -85,B 0,C 180,E1 -11959.929,E2 -11959.929} C_VEL
LIN {X 0,Y 381.746,Z 604.217,A -85,B 0,C 180,E1 -11961.528,E2 -11961.528} C_VEL
LIN {X 0,Y 381.648,Z 608.037,A -85,B 0,C 180,E1 -11963.93,E2 -11963.93} C_VEL
LIN {X 0,Y 381.573,Z 610.136,A -85,B 0,C 180,E1 -11965.773,E2 -11965.773} C_VEL
LIN {X 0,Y 381.572,Z 611.542,A -85,B 0,C 180,E1 -11967.886,E2 -11967.886} C_VEL
LIN {X 0,Y 381.634,Z 612.052,A -85,B 0,C 180,E1 -11969.997,E2 -11969.997} C_VEL
LIN {X 0,Y 381.585,Z 611.5,A -85,B 0,C 180,E1 -11972.108,E2 -11972.108} C_VEL
LIN {X 0,Y 381.571,Z 610.043,A -85,B 0,C 180,E1 -11974.222,E2 -11974.222} C_VEL
LIN {X 0,Y 381.658,Z 607.51,A -85,B 0,C 180,E1 -11976.341,E2 -11976.341} C_VEL
LIN {X 0,Y 381.743,Z 603.993,A -85,B 0,C 180,E1 -11978.467,E2 -11978.467} C_VEL
LIN {X 0,Y 381.992,Z 599.337,A -85,B 0,C 180,E1 -11980.599,E2 -11980.599} C_VEL
LIN {X 0,Y 382.581,Z 593.523,A -85,B 0,C 180,E1 -11982.732,E2 -11982.732} C_VEL
LIN {X 0,Y 383.266,Z 586.474,A -85,B 0,C 180,E1 -11984.872,E2 -11984.872} C_VEL
LIN {X 0,Y 384.588,Z 576.774,A -85,B 0,C 180,E1 -11987.271,E2 -11987.271} C_VEL
LIN {X 0,Y 385.977,Z 566.33,A -85,B 0,C 180,E1 -11989.405,E2 -11989.405} C_VEL
LIN {X 0,Y 387.606,Z 555.519,A -85,B 0,C 180,E1 -11991.259,E2 -11991.259} C_VEL
LIN {X 0,Y 389.412,Z 543.506,A -85,B 0,C 180,E1 -11993.011,E2 -11993.011} C_VEL
LIN {X 0,Y 391.303,Z 531.202,A -85,B 0,C 180,E1 -11994.537,E2 -11994.537} C_VEL
LIN {X 0,Y 393.267,Z 517.531,A -85,B 0,C 180,E1 -11995.962,E2 -11995.962} C_VEL
LIN {X 0,Y 395.228,Z 502.734,A -85,B 0,C 180,E1 -11997.24,E2 -11997.24} C_VEL
LIN {X 0,Y 397.013,Z 488.304,A -85,B 0,C 180,E1 -11998.26,E2 -11998.26} C_VEL
LIN {X 0,Y 398.648,Z 472.923,A -85,B 0,C 180,E1 -11999.141,E2 -11999.141} C_VEL
LIN {X 0,Y 399.996,Z 456.625,A -85,B 0,C 180,E1 -11999.864,E2 -11999.864} C_VEL
LIN {X 0,Y 401.204,Z 439.663,A -85,B 0,C 180,E1 -12000.381,E2 -12000.381} C_VEL
LIN {X 0,Y 402.05,Z 411.863,A -85,B 0,C 180,E1 -12000.937,E2 -12000.937} C_VEL
LIN {X 0,Y 405.888,Z 270.473,A -85,B 0,C 180,E1 -12003.573,E2 -12003.573} C_VEL
LIN {X 0,Y 403.831,Z 258.804,A -85,B 0,C 180,E1 -12004.005,E2 -12004.005} C_VEL
LIN {X 0,Y 393.155,Z 236.624,A -85,B 0,C 180,E1 -12005.491,E2 -12005.491} C_VEL
LIN {X 0,Y 389.623,Z 229.71,A -85,B 0,C 180,E1 -12006.014,E2 -12006.014} C_VEL
LIN {X 0,Y 384.323,Z 214.044,A -85,B 0,C 180,E1 -12008.835,E2 -12008.835} C_VEL
LIN {X 0,Y 382.994,Z 210.085,A -85,B 0,C 180,E1 -12009.583,E2 -12009.583} C_VEL
LIN {X 0,Y 382.985,Z 210.084,A -85,B 0,C 180,E1 -12012.776,E2 -12012.776} C_VEL
LIN {X 0,Y 382.977,Z 210.083,A -85,B 0,C 180,E1 -12015.787,E2 -12015.787} C_VEL
LIN {X 0,Y 382.992,Z 210.083,A -85,B 0,C 180,E1 -12018.789,E2 -12018.789} C_VEL
LIN {X 0,Y 382.978,Z 210.09,A -85,B 0,C 180,E1 -12022.093,E2 -12022.093} C_VEL
LIN {X 0,Y 382.992,Z 210.093,A -85,B 0,C 180,E1 -12025.33,E2 -12025.33} C_VEL
LIN {X 0,Y 382.955,Z 210.084,A -85,B 0,C 180,E1 -12029.079,E2 -12029.079} C_VEL
LIN {X 0,Y 383.028,Z 210.074,A -85,B 0,C 180,E1 -12032.696,E2 -12032.696} C_VEL
LIN {X 0,Y 383.014,Z 210.086,A -85,B 0,C 180,E1 -12036.192,E2 -12036.192} C_VEL
LIN {X 0,Y 383.052,Z 210.062,A -85,B 0,C 180,E1 -12039.599,E2 -12039.599} C_VEL
LIN {X 0,Y 383.074,Z 210.078,A -85,B 0,C 180,E1 -12042.93,E2 -12042.93} C_VEL
LIN {X 0,Y 383.095,Z 210.057,A -85,B 0,C 180,E1 -12046.463,E2 -12046.463} C_VEL
LIN {X 0,Y 383.11,Z 210.061,A -85,B 0,C 180,E1 -12049.43,E2 -12049.43} C_VEL
LIN {X 0,Y 383.227,Z 210.062,A -85,B 0,C 180,E1 -12052.625,E2 -12052.625} C_VEL
LIN {X 0,Y 383.173,Z 210.046,A -85,B 0,C 180,E1 -12054.739,E2 -12054.739} C_VEL
LIN {X 0,Y 383.356,Z 210.025,A -85,B 0,C 180,E1 -12057.899,E2 -12057.899} C_VEL
LIN {X 0,Y 383.489,Z 210.024,A -85,B 0,C 180,E1 -12060.001,E2 -12060.001} C_VEL
LIN {X 0,Y 383.22,Z 210.049,A -85,B 0,C 180,E1 -12063.154,E2 -12063.154} C_VEL
LIN {X 0,Y 383.228,Z 210.051,A -85,B 0,C 180,E1 -12066.685,E2 -12066.685} C_VEL
LIN {X 0,Y 383.121,Z 210.067,A -85,B 0,C 180,E1 -12069.503,E2 -12069.503} C_VEL
LIN {X 0,Y 383.096,Z 210.068,A -85,B 0,C 180,E1 -12073.538,E2 -12073.538} C_VEL
LIN {X 0,Y 383.067,Z 210.069,A -85,B 0,C 180,E1 -12077.457,E2 -12077.457} C_VEL
LIN {X 0,Y 383.001,Z 210.08,A -85,B 0,C 180,E1 -12080.649,E2 -12080.649} C_VEL
LIN {X 0,Y 383.007,Z 210.085,A -85,B 0,C 180,E1 -12083.81,E2 -12083.81} C_VEL
LIN {X 0,Y 383.054,Z 210.063,A -85,B 0,C 180,E1 -12086.126,E2 -12086.126} C_VEL
LIN {X 0,Y 382.967,Z 210.092,A -85,B 0,C 180,E1 -12089.703,E2 -12089.703} C_VEL
LIN {X 0,Y 382.98,Z 210.075,A -85,B 0,C 180,E1 -12093.404,E2 -12093.404} C_VEL
LIN {X 0,Y 383.01,Z 210.09,A -85,B 0,C 180,E1 -12096.167,E2 -12096.167} C_VEL
LIN {X 0,Y 382.988,Z 210.075,A -85,B 0,C 180,E1 -12099.962,E2 -12099.962} C_VEL
LIN {X 0,Y 382.988,Z 210.089,A -85,B 0,C 180,E1 -12102.782,E2 -12102.782} C_VEL
LIN {X 0,Y 382.98,Z 210.077,A -85,B 0,C 180,E1 -12105.792,E2 -12105.792} C_VEL
LIN {X 0,Y 382.959,Z 210.091,A -85,B 0,C 180,E1 -12108.802,E2 -12108.802} C_VEL
LIN {X 0,Y 382.985,Z 210.088,A -85,B 0,C 180,E1 -12112.1,E2 -12112.1} C_VEL
LIN {X 0,Y 383.007,Z 210.076,A -85,B 0,C 180,E1 -12115.336,E2 -12115.336} C_VEL
LIN {X 0,Y 382.973,Z 210.088,A -85,B 0,C 180,E1 -12119.085,E2 -12119.085} C_VEL
LIN {X 0,Y 382.986,Z 210.089,A -85,B 0,C 180,E1 -12122.697,E2 -12122.697} C_VEL
LIN {X 0,Y 383.009,Z 210.089,A -85,B 0,C 180,E1 -12126.195,E2 -12126.195} C_VEL
LIN {X 0,Y 383.052,Z 210.086,A -85,B 0,C 180,E1 -12129.602,E2 -12129.602} C_VEL
LIN {X 0,Y 383.068,Z 210.081,A -85,B 0,C 180,E1 -12132.933,E2 -12132.933} C_VEL
LIN {X 0,Y 383.126,Z 210.072,A -85,B 0,C 180,E1 -12136.467,E2 -12136.467} C_VEL
LIN {X 0,Y 383.17,Z 210.257,A -85,B 0,C 180,E1 -12140.235,E2 -12140.235} C_VEL
LIN {X 0,Y 383.572,Z 211.761,A -85,B 0,C 180,E1 -12140.46,E2 -12140.46} C_VEL
LIN {X 0,Y 392.854,Z 228.212,A -85,B 0,C 180,E1 -12141.781,E2 -12141.781} C_VEL
LIN {X 0,Y 405.856,Z 254.509,A -85,B 0,C 180,E1 -12143.57,E2 -12143.57} C_VEL
LIN {X 0,Y 405.985,Z 258.025,A -85,B 0,C 180,E1 -12143.657,E2 -12143.657} C_VEL
LIN {X 0,Y 401.588,Z 416.591,A -85,B 0,C 180,E1 -12146.63,E2 -12146.63} C_VEL
LIN {X 0,Y 400.68,Z 433.508,A -85,B 0,C 180,E1 -12147.143,E2 -12147.143} C_VEL
LIN {X 0,Y 399.511,Z 448.931,A -85,B 0,C 180,E1 -12147.797,E2 -12147.797} C_VEL
LIN {X 0,Y 398.079,Z 463.897,A -85,B 0,C 180,E1 -12148.611,E2 -12148.611} C_VEL
LIN {X 0,Y 397.543,Z 469.211,A -85,B 0,C 180,E1 -12148.954,E2 -12148.954} C_VEL
LIN {X 0,Y 396.339,Z 474.59,A -85,B 0,C 180,E1 -12149.268,E2 -12149.268} C_VEL
LIN {X 0,Y 392.685,Z 483.284,A -85,B 0,C 180,E1 -12149.726,E2 -12149.726} C_VEL
LIN {X 0,Y 388.984,Z 491.701,A -85,B 0,C 180,E1 -12150.266,E2 -12150.266} C_VEL
LIN {X 0,Y 387.717,Z 496.637,A -85,B 0,C 180,E1 -12150.703,E2 -12150.703} C_VEL
LIN {X 0,Y 385.645,Z 510.86,A -85,B 0,C 180,E1 -12152.222,E2 -12152.222} C_VEL
LIN {X 0,Y 383.783,Z 522.312,A -85,B 0,C 180,E1 -12153.677,E2 -12153.677} C_VEL
LIN {X 0,Y 381.872,Z 534.265,A -85,B 0,C 180,E1 -12155.457,E2 -12155.457} C_VEL
LIN {X 0,Y 380.25,Z 544.133,A -85,B 0,C 180,E1 -12157.169,E2 -12157.169} C_VEL
LIN {X 0,Y 378.58,Z 554.671,A -85,B 0,C 180,E1 -12159.351,E2 -12159.351} C_VEL
LIN {X 0,Y 377.231,Z 563.523,A -85,B 0,C 180,E1 -12161.555,E2 -12161.555} C_VEL
LIN {X 0,Y 376.26,Z 570.865,A -85,B 0,C 180,E1 -12163.761,E2 -12163.761} C_VEL
LIN {X 0,Y 375.541,Z 576.371,A -85,B 0,C 180,E1 -12165.747,E2 -12165.747} C_VEL
LIN {X 0,Y 375.032,Z 581.377,A -85,B 0,C 180,E1 -12168.013,E2 -12168.013} C_VEL
LIN {X 0,Y 374.649,Z 585.267,A -85,B 0,C 180,E1 -12170.289,E2 -12170.289} C_VEL
LIN {X 0,Y 374.304,Z 588.462,A -85,B 0,C 180,E1 -12173.067,E2 -12173.067} C_VEL
LIN {X 0,Y 374.234,Z 589.992,A -85,B 0,C 180,E1 -12175.652,E2 -12175.652} C_VEL
LIN {X 0,Y 374.272,Z 590.127,A -85,B 0,C 180,E1 -12178.046,E2 -12178.046} C_VEL
LIN {X 0,Y 374.339,Z 589.121,A -85,B 0,C 180,E1 -12180.46,E2 -12180.46} C_VEL
LIN {X 0,Y 374.539,Z 586.826,A -85,B 0,C 180,E1 -12182.969,E2 -12182.969} C_VEL
LIN {X 0,Y 374.953,Z 583.063,A -85,B 0,C 180,E1 -12185.526,E2 -12185.526} C_VEL
LIN {X 0,Y 375.6,Z 577.709,A -85,B 0,C 180,E1 -12188.134,E2 -12188.134} C_VEL
LIN {X 0,Y 376.359,Z 571.85,A -85,B 0,C 180,E1 -12190.357,E2 -12190.357} C_VEL
LIN {X 0,Y 377.311,Z 565.114,A -85,B 0,C 180,E1 -12192.472,E2 -12192.472} C_VEL
LIN {X 0,Y 378.798,Z 555.929,A -85,B 0,C 180,E1 -12194.833,E2 -12194.833} C_VEL
LIN {X 0,Y 380.537,Z 546.214,A -85,B 0,C 180,E1 -12196.894,E2 -12196.894} C_VEL
LIN {X 0,Y 382.432,Z 535.074,A -85,B 0,C 180,E1 -12198.892,E2 -12198.892} C_VEL
LIN {X 0,Y 384.6,Z 522.732,A -85,B 0,C 180,E1 -12200.747,E2 -12200.747} C_VEL
LIN {X 0,Y 386.855,Z 509.252,A -85,B 0,C 180,E1 -12202.443,E2 -12202.443} C_VEL
LIN {X 0,Y 388.996,Z 495.821,A -85,B 0,C 180,E1 -12203.856,E2 -12203.856} C_VEL
LIN {X 0,Y 391.09,Z 480.958,A -85,B 0,C 180,E1 -12205.152,E2 -12205.152} C_VEL
LIN {X 0,Y 392.951,Z 465.872,A -85,B 0,C 180,E1 -12206.22,E2 -12206.22} C_VEL
LIN {X 0,Y 394.508,Z 450.903,A -85,B 0,C 180,E1 -12207.071,E2 -12207.071} C_VEL
LIN {X 0,Y 395.904,Z 434.448,A -85,B 0,C 180,E1 -12207.788,E2 -12207.788} C_VEL
LIN {X 0,Y 396.906,Z 418.005,A -85,B 0,C 180,E1 -12208.3,E2 -12208.3} C_VEL
LIN {X 0,Y 401.923,Z 258.508,A -85,B 0,C 180,E1 -12211.388,E2 -12211.388} C_VEL
LIN {X 0,Y 394.45,Z 243.418,A -85,B 0,C 180,E1 -12212.554,E2 -12212.554} C_VEL
LIN {X 0,Y 385.438,Z 227.221,A -85,B 0,C 180,E1 -12214.011,E2 -12214.011} C_VEL
LIN {X 0,Y 379.05,Z 216.952,A -85,B 0,C 180,E1 -12215.087,E2 -12215.087} C_VEL
LIN {X 0,Y 376.554,Z 212.93,A -85,B 0,C 180,E1 -12215.536,E2 -12215.536} C_VEL
LIN {X 0,Y 375.994,Z 210.958,A -85,B 0,C 180,E1 -12215.995,E2 -12215.995} C_VEL
LIN {X 0,Y 375.984,Z 210.955,A -85,B 0,C 180,E1 -12219.197,E2 -12219.197} C_VEL
LIN {X 0,Y 376.054,Z 210.943,A -85,B 0,C 180,E1 -12222.601,E2 -12222.601} C_VEL
LIN {X 0,Y 376.093,Z 210.951,A -85,B 0,C 180,E1 -12226.342,E2 -12226.342} C_VEL
LIN {X 0,Y 376.121,Z 210.948,A -85,B 0,C 180,E1 -12230.318,E2 -12230.318} C_VEL
LIN {X 0,Y 376.241,Z 210.93,A -85,B 0,C 180,E1 -12233.564,E2 -12233.564} C_VEL
LIN {X 0,Y 376.351,Z 210.919,A -85,B 0,C 180,E1 -12237.859,E2 -12237.859} C_VEL
LIN {X 0,Y 376.487,Z 210.902,A -85,B 0,C 180,E1 -12239.999,E2 -12239.999} C_VEL
LIN {X 0,Y 376.183,Z 210.939,A -85,B 0,C 180,E1 -12243.212,E2 -12243.212} C_VEL
LIN {X 0,Y 376.228,Z 210.931,A -85,B 0,C 180,E1 -12246.435,E2 -12246.435} C_VEL
LIN {X 0,Y 376.114,Z 210.944,A -85,B 0,C 180,E1 -12249.681,E2 -12249.681} C_VEL
LIN {X 0,Y 376.091,Z 210.947,A -85,B 0,C 180,E1 -12253.657,E2 -12253.657} C_VEL
LIN {X 0,Y 376.034,Z 210.959,A -85,B 0,C 180,E1 -12257.399,E2 -12257.399} C_VEL
LIN {X 0,Y 375.98,Z 210.965,A -85,B 0,C 180,E1 -12260.831,E2 -12260.831} C_VEL
LIN {X 0,Y 375.991,Z 210.957,A -85,B 0,C 180,E1 -12264.281,E2 -12264.281} C_VEL
LIN {X 0,Y 376.021,Z 210.957,A -85,B 0,C 180,E1 -12266.651,E2 -12266.651} C_VEL
LIN {X 0,Y 375.965,Z 210.964,A -85,B 0,C 180,E1 -12270.312,E2 -12270.312} C_VEL
LIN {X 0,Y 375.96,Z 210.963,A -85,B 0,C 180,E1 -12274.111,E2 -12274.111} C_VEL
LIN {X 0,Y 375.954,Z 210.965,A -85,B 0,C 180,E1 -12276.741,E2 -12276.741} C_VEL
LIN {X 0,Y 375.959,Z 210.966,A -85,B 0,C 180,E1 -12279.964,E2 -12279.964} C_VEL
LIN {X 0,Y 375.93,Z 210.969,A -85,B 0,C 180,E1 -12283.765,E2 -12283.765} C_VEL
LIN {X 0,Y 375.936,Z 210.97,A -85,B 0,C 180,E1 -12286.81,E2 -12286.81} C_VEL
LIN {X 0,Y 375.948,Z 211.111,A -85,B 0,C 180,E1 -12288.612,E2 -12288.612} C_VEL
LIN {X 0,Y 381.159,Z 224.971,A -85,B 0,C 180,E1 -12291.593,E2 -12291.593} C_VEL
LIN {X 0,Y 382.509,Z 228.727,A -85,B 0,C 180,E1 -12292.298,E2 -12292.298} C_VEL
LIN {X 0,Y 391.918,Z 245.807,A -85,B 0,C 180,E1 -12293.852,E2 -12293.852} C_VEL
LIN {X 0,Y 400.388,Z 263.386,A -85,B 0,C 180,E1 -12295.198,E2 -12295.198} C_VEL
LIN {X 0,Y 401.648,Z 272.31,A -85,B 0,C 180,E1 -12295.534,E2 -12295.534} C_VEL
LIN {X 0,Y 396.518,Z 437.08,A -85,B 0,C 180,E1 -12298.72,E2 -12298.72} C_VEL
LIN {X 0,Y 395.281,Z 453.679,A -85,B 0,C 180,E1 -12299.22,E2 -12299.22} C_VEL
LIN {X 0,Y 393.873,Z 469.057,A -85,B 0,C 180,E1 -12299.876,E2 -12299.876} C_VEL
LIN {X 0,Y 392.129,Z 484.988,A -85,B 0,C 180,E1 -12300.763,E2 -12300.763} C_VEL
LIN {X 0,Y 390.189,Z 499.722,A -85,B 0,C 180,E1 -12301.782,E2 -12301.782} C_VEL
LIN {X 0,Y 387.964,Z 514.793,A -85,B 0,C 180,E1 -12303.07,E2 -12303.07} C_VEL
LIN {X 0,Y 385.727,Z 528.635,A -85,B 0,C 180,E1 -12304.502,E2 -12304.502} C_VEL
LIN {X 0,Y 383.74,Z 540.491,A -85,B 0,C 180,E1 -12305.951,E2 -12305.951} C_VEL
LIN {X 0,Y 381.897,Z 551.694,A -85,B 0,C 180,E1 -12307.549,E2 -12307.549} C_VEL
LIN {X 0,Y 379.967,Z 562.847,A -85,B 0,C 180,E1 -12309.423,E2 -12309.423} C_VEL
LIN {X 0,Y 378.219,Z 573.685,A -85,B 0,C 180,E1 -12311.583,E2 -12311.583} C_VEL
LIN {X 0,Y 376.899,Z 582.813,A -85,B 0,C 180,E1 -12313.755,E2 -12313.755} C_VEL
LIN {X 0,Y 375.935,Z 590.486,A -85,B 0,C 180,E1 -12315.932,E2 -12315.932} C_VEL
LIN {X 0,Y 375.239,Z 596.744,A -85,B 0,C 180,E1 -12318.108,E2 -12318.108} C_VEL
LIN {X 0,Y 374.766,Z 601.867,A -85,B 0,C 180,E1 -12320.281,E2 -12320.281} C_VEL
LIN {X 0,Y 374.615,Z 605.874,A -85,B 0,C 180,E1 -12322.452,E2 -12322.452} C_VEL
LIN {X 0,Y 374.486,Z 608.813,A -85,B 0,C 180,E1 -12324.613,E2 -12324.613} C_VEL
LIN {X 0,Y 374.435,Z 610.765,A -85,B 0,C 180,E1 -12326.77,E2 -12326.77} C_VEL
LIN {X 0,Y 374.517,Z 611.702,A -85,B 0,C 180,E1 -12328.922,E2 -12328.922} C_VEL
LIN {X 0,Y 374.519,Z 611.692,A -85,B 0,C 180,E1 -12331.073,E2 -12331.073} C_VEL
LIN {X 0,Y 374.434,Z 610.665,A -85,B 0,C 180,E1 -12333.225,E2 -12333.225} C_VEL
LIN {X 0,Y 374.487,Z 608.686,A -85,B 0,C 180,E1 -12335.381,E2 -12335.381} C_VEL
LIN {X 0,Y 374.611,Z 605.641,A -85,B 0,C 180,E1 -12337.543,E2 -12337.543} C_VEL
LIN {X 0,Y 374.763,Z 601.588,A -85,B 0,C 180,E1 -12339.714,E2 -12339.714} C_VEL
LIN {X 0,Y 375.391,Z 594.871,A -85,B 0,C 180,E1 -12342.43,E2 -12342.43} C_VEL
LIN {X 0,Y 376.071,Z 588.046,A -85,B 0,C 180,E1 -12344.61,E2 -12344.61} C_VEL
LIN {X 0,Y 377.19,Z 579.872,A -85,B 0,C 180,E1 -12346.783,E2 -12346.783} C_VEL
LIN {X 0,Y 378.553,Z 570.151,A -85,B 0,C 180,E1 -12348.948,E2 -12348.948} C_VEL
LIN {X 0,Y 380.111,Z 560.03,A -85,B 0,C 180,E1 -12350.846,E2 -12350.846} C_VEL
LIN {X 0,Y 382.03,Z 548.157,A -85,B 0,C 180,E1 -12352.722,E2 -12352.722} C_VEL
LIN {X 0,Y 383.784,Z 536.251,A -85,B 0,C 180,E1 -12354.329,E2 -12354.329} C_VEL
LIN {X 0,Y 385.864,Z 523.592,A -85,B 0,C 180,E1 -12355.772,E2 -12355.772} C_VEL
LIN {X 0,Y 388.075,Z 508.29,A -85,B 0,C 180,E1 -12357.227,E2 -12357.227} C_VEL
LIN {X 0,Y 390.005,Z 493.473,A -85,B 0,C 180,E1 -12358.374,E2 -12358.374} C_VEL
LIN {X 0,Y 391.813,Z 478.138,A -85,B 0,C 180,E1 -12359.33,E2 -12359.33} C_VEL
LIN {X 0,Y 393.309,Z 461.93,A -85,B 0,C 180,E1 -12360.129,E2 -12360.129} C_VEL
LIN {X 0,Y 394.554,Z 446.49,A -85,B 0,C 180,E1 -12360.689,E2 -12360.689} C_VEL
LIN {X 0,Y 395.477,Z 429.029,A -85,B 0,C 180,E1 -12361.112,E2 -12361.112} C_VEL
LIN {X 0,Y 399.833,Z 271.267,A -85,B 0,C 180,E1 -12364.1,E2 -12364.1} C_VEL
LIN {X 0,Y 398.136,Z 261.679,A -85,B 0,C 180,E1 -12364.465,E2 -12364.465} C_VEL
LIN {X 0,Y 386.703,Z 237.956,A -85,B 0,C 180,E1 -12366.101,E2 -12366.101} C_VEL
LIN {X 0,Y 382.23,Z 229.471,A -85,B 0,C 180,E1 -12366.777,E2 -12366.777} C_VEL
LIN {X 0,Y 377.718,Z 216.163,A -85,B 0,C 180,E1 -12369.238,E2 -12369.238} C_VEL
LIN {X 0,Y 375.931,Z 210.964,A -85,B 0,C 180,E1 -12370.255,E2 -12370.255} C_VEL
LIN {X 0,Y 375.909,Z 210.973,A -85,B 0,C 180,E1 -12373.763,E2 -12373.763} C_VEL
LIN {X 0,Y 375.938,Z 210.97,A -85,B 0,C 180,E1 -12377.701,E2 -12377.701} C_VEL
LIN {X 0,Y 375.944,Z 210.966,A -85,B 0,C 180,E1 -12380.536,E2 -12380.536} C_VEL
LIN {X 0,Y 375.94,Z 210.956,A -85,B 0,C 180,E1 -12383.493,E2 -12383.493} C_VEL
LIN {X 0,Y 375.934,Z 210.969,A -85,B 0,C 180,E1 -12385.886,E2 -12385.886} C_VEL
LIN {X 0,Y 375.937,Z 210.969,A -85,B 0,C 180,E1 -12389.685,E2 -12389.685} C_VEL
LIN {X 0,Y 375.991,Z 210.943,A -85,B 0,C 180,E1 -12393.346,E2 -12393.346} C_VEL
LIN {X 0,Y 375.988,Z 210.967,A -85,B 0,C 180,E1 -12396.888,E2 -12396.888} C_VEL
LIN {X 0,Y 375.987,Z 210.937,A -85,B 0,C 180,E1 -12400.339,E2 -12400.339} C_VEL
LIN {X 0,Y 375.998,Z 210.96,A -85,B 0,C 180,E1 -12403.718,E2 -12403.718} C_VEL
LIN {X 0,Y 376.076,Z 210.921,A -85,B 0,C 180,E1 -12407.042,E2 -12407.042} C_VEL
LIN {X 0,Y 376.093,Z 210.941,A -85,B 0,C 180,E1 -12410.318,E2 -12410.318} C_VEL
LIN {X 0,Y 376.218,Z 210.926,A -85,B 0,C 180,E1 -12413.565,E2 -12413.565} C_VEL
LIN {X 0,Y 376.322,Z 210.9,A -85,B 0,C 180,E1 -12417.86,E2 -12417.86} C_VEL
LIN {X 0,Y 376.458,Z 210.9,A -85,B 0,C 180,E1 -12420.001,E2 -12420.001} C_VEL
LIN {X 0,Y 376.158,Z 210.928,A -85,B 0,C 180,E1 -12423.214,E2 -12423.214} C_VEL
LIN {X 0,Y 376.192,Z 210.928,A -85,B 0,C 180,E1 -12426.674,E2 -12426.674} C_VEL
LIN {X 0,Y 376.089,Z 210.943,A -85,B 0,C 180,E1 -12429.683,E2 -12429.683} C_VEL
LIN {X 0,Y 376.06,Z 210.945,A -85,B 0,C 180,E1 -12433.659,E2 -12433.659} C_VEL
LIN {X 0,Y 376.016,Z 210.947,A -85,B 0,C 180,E1 -12437.609,E2 -12437.609} C_VEL
LIN {X 0,Y 375.951,Z 210.961,A -85,B 0,C 180,E1 -12440.834,E2 -12440.834} C_VEL
LIN {X 0,Y 375.968,Z 210.957,A -85,B 0,C 180,E1 -12444.284,E2 -12444.284} C_VEL
LIN {X 0,Y 375.995,Z 210.945,A -85,B 0,C 180,E1 -12446.655,E2 -12446.655} C_VEL
LIN {X 0,Y 375.94,Z 210.968,A -85,B 0,C 180,E1 -12450.315,E2 -12450.315} C_VEL
LIN {X 0,Y 375.938,Z 210.957,A -85,B 0,C 180,E1 -12454.114,E2 -12454.114} C_VEL
LIN {X 0,Y 375.932,Z 210.968,A -85,B 0,C 180,E1 -12456.744,E2 -12456.744} C_VEL
LIN {X 0,Y 375.968,Z 210.949,A -85,B 0,C 180,E1 -12459.974,E2 -12459.974} C_VEL
LIN {X 0,Y 375.912,Z 210.969,A -85,B 0,C 180,E1 -12463.769,E2 -12463.769} C_VEL
LIN {X 0,Y 375.919,Z 210.97,A -85,B 0,C 180,E1 -12466.814,E2 -12466.814} C_VEL
LIN {X 0,Y 375.934,Z 210.957,A -85,B 0,C 180,E1 -12470.539,E2 -12470.539} C_VEL
LIN {X 0,Y 375.952,Z 210.967,A -85,B 0,C 180,E1 -12473.499,E2 -12473.499} C_VEL
LIN {X 0,Y 375.949,Z 210.956,A -85,B 0,C 180,E1 -12475.892,E2 -12475.892} C_VEL
LIN {X 0,Y 375.953,Z 210.959,A -85,B 0,C 180,E1 -12479.691,E2 -12479.691} C_VEL
LIN {X 0,Y 375.928,Z 210.973,A -85,B 0,C 180,E1 -12482.14,E2 -12482.14} C_VEL
LIN {X 0,Y 375.966,Z 210.966,A -85,B 0,C 180,E1 -12485.72,E2 -12485.72} C_VEL
LIN {X 0,Y 375.995,Z 210.963,A -85,B 0,C 180,E1 -12489.201,E2 -12489.201} C_VEL
LIN {X 0,Y 376.012,Z 210.961,A -85,B 0,C 180,E1 -12492.603,E2 -12492.603} C_VEL
LIN {X 0,Y 376.09,Z 210.947,A -85,B 0,C 180,E1 -12496.346,E2 -12496.346} C_VEL
LIN {X 0,Y 376.108,Z 211.047,A -85,B 0,C 180,E1 -12499.574,E2 -12499.574} C_VEL
LIN {X 0,Y 376.324,Z 212.109,A -85,B 0,C 180,E1 -12499.695,E2 -12499.695} C_VEL
LIN {X 0,Y 377.818,Z 214.774,A -85,B 0,C 180,E1 -12499.921,E2 -12499.921} C_VEL
LIN {X 0,Y 385.633,Z 228.369,A -85,B 0,C 180,E1 -12501.059,E2 -12501.059} C_VEL
LIN {X 0,Y 392.228,Z 241.228,A -85,B 0,C 180,E1 -12502.012,E2 -12502.012} C_VEL
LIN {X 0,Y 400.007,Z 257.093,A -85,B 0,C 180,E1 -12503.095,E2 -12503.095} C_VEL
LIN {X 0,Y 395.388,Z 417.728,A -85,B 0,C 180,E1 -12506.157,E2 -12506.157} C_VEL
LIN {X 0,Y 394.39,Z 434.679,A -85,B 0,C 180,E1 -12506.686,E2 -12506.686} C_VEL
LIN {X 0,Y 393.153,Z 450.369,A -85,B 0,C 180,E1 -12507.377,E2 -12507.377} C_VEL
LIN {X 0,Y 391.652,Z 465.073,A -85,B 0,C 180,E1 -12508.203,E2 -12508.203} C_VEL
LIN {X 0,Y 390.043,Z 479.675,A -85,B 0,C 180,E1 -12509.228,E2 -12509.228} C_VEL
LIN {X 0,Y 387.986,Z 494.739,A -85,B 0,C 180,E1 -12510.521,E2 -12510.521} C_VEL
LIN {X 0,Y 387.717,Z 496.637,A -85,B 0,C 180,E1 -12510.703,E2 -12510.703} C_VEL
LIN {X 0,Y 386.438,Z 501.614,A -85,B 0,C 180,E1 -12511.163,E2 -12511.163} C_VEL
LIN {X 0,Y 382.597,Z 509.51,A -85,B 0,C 180,E1 -12511.846,E2 -12511.846} C_VEL
LIN {X 0,Y 378.697,Z 517.138,A -85,B 0,C 180,E1 -12512.589,E2 -12512.589} C_VEL
LIN {X 0,Y 377.329,Z 521.535,A -85,B 0,C 180,E1 -12513.137,E2 -12513.137} C_VEL
LIN {X 0,Y 375.445,Z 532.984,A -85,B 0,C 180,E1 -12514.834,E2 -12514.834} C_VEL
LIN {X 0,Y 373.542,Z 543.974,A -85,B 0,C 180,E1 -12516.755,E2 -12516.755} C_VEL
LIN {X 0,Y 371.759,Z 554.579,A -85,B 0,C 180,E1 -12518.975,E2 -12518.975} C_VEL
LIN {X 0,Y 370.364,Z 563.475,A -85,B 0,C 180,E1 -12521.218,E2 -12521.218} C_VEL
LIN {X 0,Y 369.405,Z 570.099,A -85,B 0,C 180,E1 -12523.199,E2 -12523.199} C_VEL
LIN {X 0,Y 368.551,Z 576.396,A -85,B 0,C 180,E1 -12525.486,E2 -12525.486} C_VEL
LIN {X 0,Y 367.99,Z 581.446,A -85,B 0,C 180,E1 -12527.795,E2 -12527.795} C_VEL
LIN {X 0,Y 367.533,Z 585.82,A -85,B 0,C 180,E1 -12530.447,E2 -12530.447} C_VEL
LIN {X 0,Y 367.255,Z 588.205,A -85,B 0,C 180,E1 -12532.505,E2 -12532.505} C_VEL
LIN {X 0,Y 367.12,Z 589.869,A -85,B 0,C 180,E1 -12534.91,E2 -12534.91} C_VEL
LIN {X 0,Y 367.135,Z 590.432,A -85,B 0,C 180,E1 -12537.352,E2 -12537.352} C_VEL
LIN {X 0,Y 367.22,Z 589.754,A -85,B 0,C 180,E1 -12539.843,E2 -12539.843} C_VEL
LIN {X 0,Y 367.379,Z 587.779,A -85,B 0,C 180,E1 -12542.389,E2 -12542.389} C_VEL
LIN {X 0,Y 367.745,Z 584.433,A -85,B 0,C 180,E1 -12544.985,E2 -12544.985} C_VEL
LIN {X 0,Y 368.355,Z 579.555,A -85,B 0,C 180,E1 -12547.63,E2 -12547.63} C_VEL
LIN {X 0,Y 369.006,Z 574.765,A -85,B 0,C 180,E1 -12549.647,E2 -12549.647} C_VEL
LIN {X 0,Y 369.883,Z 568.919,A -85,B 0,C 180,E1 -12551.685,E2 -12551.685} C_VEL
LIN {X 0,Y 371.182,Z 560.982,A -85,B 0,C 180,E1 -12553.986,E2 -12553.986} C_VEL
LIN {X 0,Y 372.843,Z 551.936,A -85,B 0,C 180,E1 -12556.139,E2 -12556.139} C_VEL
LIN {X 0,Y 374.716,Z 541.409,A -85,B 0,C 180,E1 -12558.248,E2 -12558.248} C_VEL
LIN {X 0,Y 376.899,Z 529.665,A -85,B 0,C 180,E1 -12560.218,E2 -12560.218} C_VEL
LIN {X 0,Y 379.166,Z 517.174,A -85,B 0,C 180,E1 -12561.977,E2 -12561.977} C_VEL
LIN {X 0,Y 381.37,Z 504.324,A -85,B 0,C 180,E1 -12563.509,E2 -12563.509} C_VEL
LIN {X 0,Y 383.509,Z 490.654,A -85,B 0,C 180,E1 -12564.864,E2 -12564.864} C_VEL
LIN {X 0,Y 385.586,Z 476.032,A -85,B 0,C 180,E1 -12566.065,E2 -12566.065} C_VEL
LIN {X 0,Y 387.361,Z 461.817,A -85,B 0,C 180,E1 -12567.023,E2 -12567.023} C_VEL
LIN {X 0,Y 389.032,Z 445.409,A -85,B 0,C 180,E1 -12567.899,E2 -12567.899} C_VEL
LIN {X 0,Y 390.356,Z 428.423,A -85,B 0,C 180,E1 -12568.567,E2 -12568.567} C_VEL
LIN {X 0,Y 391.213,Z 412.334,A -85,B 0,C 180,E1 -12568.991,E2 -12568.991} C_VEL
LIN {X 0,Y 396.197,Z 260.806,A -85,B 0,C 180,E1 -12571.952,E2 -12571.952} C_VEL
LIN {X 0,Y 387.817,Z 244.148,A -85,B 0,C 180,E1 -12573.305,E2 -12573.305} C_VEL
LIN {X 0,Y 379.969,Z 230.209,A -85,B 0,C 180,E1 -12574.625,E2 -12574.625} C_VEL
LIN {X 0,Y 372.121,Z 217.604,A -85,B 0,C 180,E1 -12576.01,E2 -12576.01} C_VEL
LIN {X 0,Y 369.458,Z 213.741,A -85,B 0,C 180,E1 -12576.491,E2 -12576.491} C_VEL
LIN {X 0,Y 368.978,Z 211.963,A -85,B 0,C 180,E1 -12576.83,E2 -12576.83} C_VEL
LIN {X 0,Y 368.934,Z 211.836,A -85,B 0,C 180,E1 -12579.946,E2 -12579.946} C_VEL
LIN {X 0,Y 368.979,Z 211.829,A -85,B 0,C 180,E1 -12583.398,E2 -12583.398} C_VEL
LIN {X 0,Y 369.061,Z 211.824,A -85,B 0,C 180,E1 -12586.79,E2 -12586.79} C_VEL
LIN {X 0,Y 369.069,Z 211.826,A -85,B 0,C 180,E1 -12590.131,E2 -12590.131} C_VEL
LIN {X 0,Y 369.201,Z 211.808,A -85,B 0,C 180,E1 -12593.441,E2 -12593.441} C_VEL
LIN {X 0,Y 369.316,Z 211.796,A -85,B 0,C 180,E1 -12597.818,E2 -12597.818} C_VEL
LIN {X 0,Y 369.457,Z 211.778,A -85,B 0,C 180,E1 -12599.999,E2 -12599.999} C_VEL
LIN {X 0,Y 369.316,Z 211.791,A -85,B 0,C 180,E1 -12602.181,E2 -12602.181} C_VEL
LIN {X 0,Y 369.187,Z 211.808,A -85,B 0,C 180,E1 -12606.558,E2 -12606.558} C_VEL
LIN {X 0,Y 369.064,Z 211.82,A -85,B 0,C 180,E1 -12609.868,E2 -12609.868} C_VEL
LIN {X 0,Y 369.039,Z 211.826,A -85,B 0,C 180,E1 -12613.771,E2 -12613.771} C_VEL
LIN {X 0,Y 368.993,Z 211.834,A -85,B 0,C 180,E1 -12617.742,E2 -12617.742} C_VEL
LIN {X 0,Y 368.912,Z 211.842,A -85,B 0,C 180,E1 -12621.22,E2 -12621.22} C_VEL
LIN {X 0,Y 368.957,Z 211.833,A -85,B 0,C 180,E1 -12624.775,E2 -12624.775} C_VEL
LIN {X 0,Y 368.964,Z 211.834,A -85,B 0,C 180,E1 -12627.203,E2 -12627.203} C_VEL
LIN {X 0,Y 368.915,Z 211.846,A -85,B 0,C 180,E1 -12630.954,E2 -12630.954} C_VEL
LIN {X 0,Y 368.937,Z 211.839,A -85,B 0,C 180,E1 -12634.853,E2 -12634.853} C_VEL
LIN {X 0,Y 368.907,Z 211.843,A -85,B 0,C 180,E1 -12638.638,E2 -12638.638} C_VEL
LIN {X 0,Y 368.876,Z 211.841,A -85,B 0,C 180,E1 -12642.007,E2 -12642.007} C_VEL
LIN {X 0,Y 368.879,Z 211.842,A -85,B 0,C 180,E1 -12645.174,E2 -12645.174} C_VEL
LIN {X 0,Y 368.901,Z 211.978,A -85,B 0,C 180,E1 -12647.727,E2 -12647.727} C_VEL
LIN {X 0,Y 374.302,Z 226.177,A -85,B 0,C 180,E1 -12650.911,E2 -12650.911} C_VEL
LIN {X 0,Y 375.141,Z 228.388,A -85,B 0,C 180,E1 -12651.331,E2 -12651.331} C_VEL
LIN {X 0,Y 384.042,Z 244.219,A -85,B 0,C 180,E1 -12652.878,E2 -12652.878} C_VEL
LIN {X 0,Y 391.435,Z 258.788,A -85,B 0,C 180,E1 -12654.108,E2 -12654.108} C_VEL
LIN {X 0,Y 394.974,Z 266.675,A -85,B 0,C 180,E1 -12654.688,E2 -12654.688} C_VEL
LIN {X 0,Y 395.919,Z 273.314,A -85,B 0,C 180,E1 -12654.946,E2 -12654.946} C_VEL
LIN {X 0,Y 390.582,Z 436.557,A -85,B 0,C 180,E1 -12658.149,E2 -12658.149} C_VEL
LIN {X 0,Y 389.306,Z 453.299,A -85,B 0,C 180,E1 -12658.657,E2 -12658.657} C_VEL
LIN {X 0,Y 387.873,Z 468.077,A -85,B 0,C 180,E1 -12659.285,E2 -12659.285} C_VEL
LIN {X 0,Y 386.199,Z 483.194,A -85,B 0,C 180,E1 -12660.12,E2 -12660.12} C_VEL
LIN {X 0,Y 384.171,Z 498.109,A -85,B 0,C 180,E1 -12661.149,E2 -12661.149} C_VEL
LIN {X 0,Y 381.92,Z 512.912,A -85,B 0,C 180,E1 -12662.41,E2 -12662.41} C_VEL
LIN {X 0,Y 379.447,Z 527.42,A -85,B 0,C 180,E1 -12663.901,E2 -12663.901} C_VEL
LIN {X 0,Y 377.184,Z 540.426,A -85,B 0,C 180,E1 -12665.505,E2 -12665.505} C_VEL
LIN {X 0,Y 375.28,Z 551.619,A -85,B 0,C 180,E1 -12667.131,E2 -12667.131} C_VEL
LIN {X 0,Y 373.245,Z 562.75,A -85,B 0,C 180,E1 -12669.035,E2 -12669.035} C_VEL
LIN {X 0,Y 371.527,Z 572.753,A -85,B 0,C 180,E1 -12671.053,E2 -12671.053} C_VEL
LIN {X 0,Y 370.193,Z 581.647,A -85,B 0,C 180,E1 -12673.169,E2 -12673.169} C_VEL
LIN {X 0,Y 368.959,Z 590.325,A -85,B 0,C 180,E1 -12675.661,E2 -12675.661} C_VEL
LIN {X 0,Y 368.207,Z 596.579,A -85,B 0,C 180,E1 -12677.878,E2 -12677.878} C_VEL
LIN {X 0,Y 367.688,Z 601.691,A -85,B 0,C 180,E1 -12680.092,E2 -12680.092} C_VEL
LIN {X 0,Y 367.532,Z 605.696,A -85,B 0,C 180,E1 -12682.305,E2 -12682.305} C_VEL
LIN {X 0,Y 367.408,Z 608.625,A -85,B 0,C 180,E1 -12684.509,E2 -12684.509} C_VEL
LIN {X 0,Y 367.351,Z 610.573,A -85,B 0,C 180,E1 -12686.707,E2 -12686.707} C_VEL
LIN {X 0,Y 367.418,Z 611.499,A -85,B 0,C 180,E1 -12688.901,E2 -12688.901} C_VEL
LIN {X 0,Y 367.419,Z 611.484,A -85,B 0,C 180,E1 -12691.093,E2 -12691.093} C_VEL
LIN {X 0,Y 367.351,Z 610.446,A -85,B 0,C 180,E1 -12693.288,E2 -12693.288} C_VEL
LIN {X 0,Y 367.408,Z 608.46,A -85,B 0,C 180,E1 -12695.485,E2 -12695.485} C_VEL
LIN {X 0,Y 367.528,Z 605.399,A -85,B 0,C 180,E1 -12697.69,E2 -12697.69} C_VEL
LIN {X 0,Y 367.684,Z 601.335,A -85,B 0,C 180,E1 -12699.903,E2 -12699.903} C_VEL
LIN {X 0,Y 368.384,Z 594.6,A -85,B 0,C 180,E1 -12702.67,E2 -12702.67} C_VEL
LIN {X 0,Y 369.09,Z 587.756,A -85,B 0,C 180,E1 -12704.892,E2 -12704.892} C_VEL
LIN {X 0,Y 370.305,Z 579.562,A -85,B 0,C 180,E1 -12707.105,E2 -12707.105} C_VEL
LIN {X 0,Y 371.701,Z 569.78,A -85,B 0,C 180,E1 -12709.318,E2 -12709.318} C_VEL
LIN {X 0,Y 373.375,Z 559.68,A -85,B 0,C 180,E1 -12711.24,E2 -12711.24} C_VEL
LIN {X 0,Y 375.386,Z 547.776,A -85,B 0,C 180,E1 -12713.148,E2 -12713.148} C_VEL
LIN {X 0,Y 377.282,Z 535.838,A -85,B 0,C 180,E1 -12714.776,E2 -12714.776} C_VEL
LIN {X 0,Y 379.378,Z 523.123,A -85,B 0,C 180,E1 -12716.246,E2 -12716.246} C_VEL
LIN {X 0,Y 381.607,Z 508.31,A -85,B 0,C 180,E1 -12717.674,E2 -12717.674} C_VEL
LIN {X 0,Y 383.722,Z 492.873,A -85,B 0,C 180,E1 -12718.882,E2 -12718.882} C_VEL
LIN {X 0,Y 385.542,Z 477.405,A -85,B 0,C 180,E1 -12719.855,E2 -12719.855} C_VEL
LIN {X 0,Y 387.118,Z 460.998,A -85,B 0,C 180,E1 -12720.662,E2 -12720.662} C_VEL
LIN {X 0,Y 388.444,Z 445.2,A -85,B 0,C 180,E1 -12721.225,E2 -12721.225} C_VEL
LIN {X 0,Y 389.305,Z 427.894,A -85,B 0,C 180,E1 -12721.646,E2 -12721.646} C_VEL
LIN {X 0,Y 393.842,Z 272.783,A -85,B 0,C 180,E1 -12724.621,E2 -12724.621} C_VEL
LIN {X 0,Y 392.446,Z 264.573,A -85,B 0,C 180,E1 -12724.935,E2 -12724.935} C_VEL
LIN {X 0,Y 381.596,Z 242.034,A -85,B 0,C 180,E1 -12726.53,E2 -12726.53} C_VEL
LIN {X 0,Y 374.921,Z 229.324,A -85,B 0,C 180,E1 -12727.549,E2 -12727.549} C_VEL
LIN {X 0,Y 370.78,Z 217.227,A -85,B 0,C 180,E1 -12729.857,E2 -12729.857} C_VEL
LIN {X 0,Y 368.878,Z 211.848,A -85,B 0,C 180,E1 -12730.945,E2 -12730.945} C_VEL
LIN {X 0,Y 368.859,Z 211.847,A -85,B 0,C 180,E1 -12734.821,E2 -12734.821} C_VEL
LIN {X 0,Y 368.887,Z 211.845,A -85,B 0,C 180,E1 -12738.179,E2 -12738.179} C_VEL
LIN {X 0,Y 368.889,Z 211.849,A -85,B 0,C 180,E1 -12741.357,E2 -12741.357} C_VEL
LIN {X 0,Y 368.911,Z 211.844,A -85,B 0,C 180,E1 -12745.144,E2 -12745.144} C_VEL
LIN {X 0,Y 368.886,Z 211.835,A -85,B 0,C 180,E1 -12749.043,E2 -12749.043} C_VEL
LIN {X 0,Y 368.935,Z 211.826,A -85,B 0,C 180,E1 -12752.795,E2 -12752.795} C_VEL
LIN {X 0,Y 368.951,Z 211.839,A -85,B 0,C 180,E1 -12756.421,E2 -12756.421} C_VEL
LIN {X 0,Y 368.926,Z 211.817,A -85,B 0,C 180,E1 -12759.947,E2 -12759.947} C_VEL
LIN {X 0,Y 368.946,Z 211.84,A -85,B 0,C 180,E1 -12763.398,E2 -12763.398} C_VEL
LIN {X 0,Y 369.029,Z 211.801,A -85,B 0,C 180,E1 -12766.79,E2 -12766.79} C_VEL
LIN {X 0,Y 369.042,Z 211.818,A -85,B 0,C 180,E1 -12770.132,E2 -12770.132} C_VEL
LIN {X 0,Y 369.134,Z 211.817,A -85,B 0,C 180,E1 -12772.342,E2 -12772.342} C_VEL
LIN {X 0,Y 369.118,Z 211.798,A -85,B 0,C 180,E1 -12774.538,E2 -12774.538} C_VEL
LIN {X 0,Y 369.287,Z 211.776,A -85,B 0,C 180,E1 -12777.819,E2 -12777.819} C_VEL
LIN {X 0,Y 369.428,Z 211.776,A -85,B 0,C 180,E1 -12780.001,E2 -12780.001} C_VEL
LIN {X 0,Y 369.287,Z 211.797,A -85,B 0,C 180,E1 -12782.182,E2 -12782.182} C_VEL
LIN {X 0,Y 369.161,Z 211.805,A -85,B 0,C 180,E1 -12786.66,E2 -12786.66} C_VEL
LIN {X 0,Y 369.037,Z 211.822,A -85,B 0,C 180,E1 -12789.87,E2 -12789.87} C_VEL
LIN {X 0,Y 369.008,Z 211.823,A -85,B 0,C 180,E1 -12793.774,E2 -12793.774} C_VEL
LIN {X 0,Y 368.974,Z 211.823,A -85,B 0,C 180,E1 -12797.77,E2 -12797.77} C_VEL
LIN {X 0,Y 368.903,Z 211.841,A -85,B 0,C 180,E1 -12801.222,E2 -12801.222} C_VEL
LIN {X 0,Y 368.932,Z 211.826,A -85,B 0,C 180,E1 -12804.778,E2 -12804.778} C_VEL
LIN {X 0,Y 368.938,Z 211.831,A -85,B 0,C 180,E1 -12807.206,E2 -12807.206} C_VEL
LIN {X 0,Y 368.894,Z 211.845,A -85,B 0,C 180,E1 -12809.693,E2 -12809.693} C_VEL
LIN {X 0,Y 368.874,Z 211.83,A -85,B 0,C 180,E1 -12813.046,E2 -12813.046} C_VEL
LIN {X 0,Y 368.896,Z 211.849,A -85,B 0,C 180,E1 -12816.2,E2 -12816.2} C_VEL
LIN {X 0,Y 368.88,Z 211.828,A -85,B 0,C 180,E1 -12818.957,E2 -12818.957} C_VEL
LIN {X 0,Y 368.863,Z 211.851,A -85,B 0,C 180,E1 -12822.013,E2 -12822.013} C_VEL
LIN {X 0,Y 368.862,Z 211.832,A -85,B 0,C 180,E1 -12825.179,E2 -12825.179} C_VEL
LIN {X 0,Y 368.86,Z 211.853,A -85,B 0,C 180,E1 -12828.18,E2 -12828.18} C_VEL
LIN {X 0,Y 368.869,Z 211.84,A -85,B 0,C 180,E1 -12831.368,E2 -12831.368} C_VEL
LIN {X 0,Y 368.926,Z 211.83,A -85,B 0,C 180,E1 -12835.15,E2 -12835.15} C_VEL
LIN {X 0,Y 368.921,Z 211.839,A -85,B 0,C 180,E1 -12839.05,E2 -12839.05} C_VEL
LIN {X 0,Y 368.865,Z 211.848,A -85,B 0,C 180,E1 -12842.793,E2 -12842.793} C_VEL
LIN {X 0,Y 368.943,Z 211.838,A -85,B 0,C 180,E1 -12846.424,E2 -12846.424} C_VEL
LIN {X 0,Y 368.931,Z 211.84,A -85,B 0,C 180,E1 -12849.95,E2 -12849.95} C_VEL
LIN {X 0,Y 368.925,Z 211.839,A -85,B 0,C 180,E1 -12853.4,E2 -12853.4} C_VEL
LIN {X 0,Y 369.058,Z 211.826,A -85,B 0,C 180,E1 -12856.793,E2 -12856.793} C_VEL
LIN {X 0,Y 369.03,Z 211.828,A -85,B 0,C 180,E1 -12858.851,E2 -12858.851} C_VEL
LIN {X 0,Y 370.107,Z 214.799,A -85,B 0,C 180,E1 -12859.068,E2 -12859.068} C_VEL
LIN {X 0,Y 371.744,Z 217.181,A -85,B 0,C 180,E1 -12859.311,E2 -12859.311} C_VEL
LIN {X 0,Y 379.091,Z 229.728,A -85,B 0,C 180,E1 -12860.412,E2 -12860.412} C_VEL
LIN {X 0,Y 386.91,Z 244.833,A -85,B 0,C 180,E1 -12861.567,E2 -12861.567} C_VEL
LIN {X 0,Y 393.865,Z 258.934,A -85,B 0,C 180,E1 -12862.564,E2 -12862.564} C_VEL
LIN {X 0,Y 391.27,Z 347.622,A -85,B 0,C 180,E1 -12864.269,E2 -12864.269} C_VEL
LIN {X 0,Y 389.227,Z 417.366,A -85,B 0,C 180,E1 -12865.634,E2 -12865.634} C_VEL
LIN {X 0,Y 388.234,Z 434.066,A -85,B 0,C 180,E1 -12866.156,E2 -12866.156} C_VEL
LIN {X 0,Y 386.987,Z 449.411,A -85,B 0,C 180,E1 -12866.826,E2 -12866.826} C_VEL
LIN {X 0,Y 385.475,Z 464.191,A -85,B 0,C 180,E1 -12867.652,E2 -12867.652} C_VEL
LIN {X 0,Y 383.803,Z 478.942,A -85,B 0,C 180,E1 -12868.691,E2 -12868.691} C_VEL
LIN {X 0,Y 381.626,Z 494.213,A -85,B 0,C 180,E1 -12870.003,E2 -12870.003} C_VEL
LIN {X 0,Y 379.629,Z 507.542,A -85,B 0,C 180,E1 -12871.394,E2 -12871.394} C_VEL
LIN {X 0,Y 377.578,Z 520.078,A -85,B 0,C 180,E1 -12872.937,E2 -12872.937} C_VEL
LIN {X 0,Y 377.329,Z 521.535,A -85,B 0,C 180,E1 -12873.137,E2 -12873.137} C_VEL
LIN {X 0,Y 375.976,Z 525.962,A -85,B 0,C 180,E1 -12873.713,E2 -12873.713} C_VEL
LIN {X 0,Y 368.883,Z 538.315,A -85,B 0,C 180,E1 -12875.377,E2 -12875.377} C_VEL
